// TwinCAT 3 PLC project PLC
// ProgramVersion: 3.1.4023.0
// libraries:
//   Tc2_Standard, * (Beckhoff Automation GmbH)
//   Tc2_System, * (Beckhoff Automation GmbH)
//   Tc3_Module, * (Beckhoff Automation GmbH)
// project tree:
//   / PlcTask.TcTTO
//   POUs/ MAIN.TcPOU
//   DUTs/IO/PDOs/ InfoData_6F19DB2B.TcDUT, CC_Inputs_2C1C9EE0.TcDUT, CC_Outputs_69F9BE14.TcDUT, WcState_9091E0EB.TcDUT, InfoData_BEF6B88E.TcDUT, FB_Inputs_4BC4AA01.TcDUT, FB_Outputs_DAFD38E0.TcDUT, InfoData_A7436BC6.TcDUT, CC_Inputs_14_Ch_F1B79554.TcDUT, CC_Outputs_14_Ch_45965511.TcDUT, FB_Inputs_39145651.TcDUT, FB_Inputs_01C60045.TcDUT, FB_Inputs_2D665851.TcDUT, InfoData_E68C61CD.TcDUT, WcState_0B2B16F9.TcDUT, InfoData_2A97D6CF.TcDUT, Inputs_25A0042B.TcDUT, Outputs_2397A10E.TcDUT
//   DUTs/IO/Boxes/ EK1100_1FC0878B.TcDUT, EK1122_1FC0878B.TcDUT, AT2020_2EA6C9BF.TcDUT, AT2050_33A3DF1B.TcDUT, AT2000_1809CD2F.TcDUT, AT2000_2EA6C9BF.TcDUT, AT2001_2EA6C9BF.TcDUT, AT2002_2EA6C9BF.TcDUT, AT2021_2EA6C9BF.TcDUT, AT2025_2EA6C9BF.TcDUT, AT2026_2EA6C9BF.TcDUT, AT2040_2EA6C9BF.TcDUT, AT2000_33A3DF1B.TcDUT, AT2026_33A3DF1B.TcDUT, AT2041_2EA6C9BF.TcDUT, AT2042_33A3DF1B.TcDUT, AT2041_33A3DF1B.TcDUT, AT2040_33A3DF1B.TcDUT, AT2042_2EA6C9BF.TcDUT, AT2025_33A3DF1B.TcDUT, AT2050_2EA6C9BF.TcDUT, AT2021_33A3DF1B.TcDUT, AT2020_33A3DF1B.TcDUT, AT2001_33A3DF1B.TcDUT, AT2002_33A3DF1B.TcDUT, ATH2000_2EA6C9BF.TcDUT, ATH2050_6EC099B7.TcDUT, ATH2040_41437DDC.TcDUT, ATH2040_2EA6C9BF.TcDUT, ATH2050_2EA6C9BF.TcDUT, ATH2000_D874080E.TcDUT
//   DUTs/IO/Devices/ SyncUnitTask_2D604ED5.TcDUT, SyncUnitTasks_6FEB8257.TcDUT, SyncUnits_99E584AF.TcDUT
//   DUTs/IO/Topology/ A_0060_AT2020_0250_0019_AT2020_0250_29EE8276.TcDUT, A_0036_AT2040_0250_0021_0B822AE4.TcDUT, A_0037_AT2040_0250_0022_033DCEC4.TcDUT, A_0038_AT2040_0250_0023_C339CA0C.TcDUT, A_0039_AT2040_0250_0024_375958EA.TcDUT, A_0040_AT2041_0250_0018_536500F2.TcDUT, A_0041_AT2041_0250_0019_F34F4056.TcDUT, A_0042_AT2041_0250_0020_5E65A51E.TcDUT, A_0043_AT2041_0250_0021_AA0537F8.TcDUT, A_0044_AT2041_0250_0022_5A9A39BA.TcDUT, A_0045_AT2041_0250_0023_51C662AC.TcDUT, A_0046_AT2042_0250_0024_1B20CF31.TcDUT, A_0047_AT2050_0500_0016_139F2B11.TcDUT, A_0048_AT2050_0500_0017_3F977F47.TcDUT, A_0049_AT2050_0500_0018_CBE655A8.TcDUT, A_0050_AT2050_0500_0019_15A3AE6F.TcDUT, A_0051_AT2050_0500_0020_9B531B4E.TcDUT, A_0052_AT2050_0500_0021_4516E089.TcDUT, A_0053_AT2050_0500_0022_433BDDFE.TcDUT, A_0054_AT2050_0500_0023_B2F2DF55.TcDUT, A_0055_AT2050_0500_0024_8D42A08D.TcDUT, A_0056_AT2050_0501_0017_A14AF4DB.TcDUT, A_0057_AT2050_0501_0020_A9F510FB.TcDUT, A_0058_AT2050_0501_0021_DD8E1090.TcDUT, A_0061_AT2020_0250_0023_AT2020_0250_2D9AB3DC.TcDUT, A_0062_AT2025_0250_0020_AT2025_0250_8DB0F378.TcDUT, A_0063_AT2025_0250_0022_AT2025_0250_E88F66A2.TcDUT, A_0064_AT2025_0250_0023_AT2025_0250_894F6FDC.TcDUT, A_0065_AT2026_0250_0019_AT2026_0250_A5473B8A.TcDUT, A_0066_AT2026_0250_0020_AT2026_0250_ADF8DFAA.TcDUT, A_0067_AT2026_0250_0022_AT2026_0250_BF728FE6.TcDUT, A_0068_AT2026_0250_0024_AT2026_0250_71C01165.TcDUT, A_0069_AT2050_0501_0019_AT2050_0501_10255FA6.TcDUT, A_0070_AT2050_0501_0022_AT2050_0501_E445CD40.TcDUT, A_0071_AT2050_0501_0023_AT2050_0501_A5CC9684.TcDUT, A_0072_AT2050_0501_0024_AT2050_0501_05E6D620.TcDUT, Beckhoff_AT2xxxEK1122_43DD63D7.TcDUT, Beckhoff_AT1xxx_27B72169.TcDUT, A_0001_ATH2000_0250_0022_300D1FD0.TcDUT, A_0002_ATH2000_0250_0023_E62B11EA.TcDUT, Beckhoff_ATH2xxxEK1122_61A38CAE.TcDUT, Beckhoff_ATH2xxx_11442560.TcDUT, EtherCAT_Master_ATxxxx_981D2C79.TcDUT
//   DUTs/IO/Base/ EtcSlaveBase_82538BE2.TcDUT, EtcSlaveBase_82538BE2.TcDUT, EtcSlaveBase_82538BE2.TcDUT, EtcSlaveTerminalBase_947E5A46.TcDUT, EtcSlaveBoxBase_77A0E4A7.TcDUT, EtcSlaveEndTerminalBase_866C7F0C.TcDUT, InputBase_8311D824.TcDUT, OutputBase_10CEE7DE.TcDUT, EtcMasterBase_62654B43.TcDUT
//   GVLs/ GVL_iXlinker.TcGVL
// real-time tasks:
//   TASK PlcTask: cycle T#10ms, priority 20, ADS port 350
// I/O:
//   DEVICE EtherCAT_Master_ATxxxx, AmsNetId 172.20.30.238.4.1
//     Beckhoff AT1xxx [EK1100 EtherCAT Coupler (2A E-Bus)]
//       Beckhoff AT2xxxEK1122 [EK1122 2 port EtherCAT junction]
//         A_0060(AT2020-0250-0019) (AT2020-0250) [AT2020-0250 Motor module, +22.5°, 250mm, 50V]
//           A_0085(AT2050-5500-0018) (AT2050-5500) [AT2050-5500 Sensor line 90° clothoid, EtherCAT In]
//         Beckhoff AT2xxxsub EK1100 [EK1100 EtherCAT Coupler (2A E-Bus)]
//         A_0001(AT2000-0233-0022) [AT2000-0233 Motor module 233 mm, 48V]
//         A_0002(AT2000-0233-0023) [AT2000-0233 Motor module 233 mm, 48V]
//         A_0003(AT2000-0233-0024) [AT2000-0233 Motor module 233 mm, 48V]
//         A_0004(AT2000-0250-0016) [AT2000-0250 Motor module 250 mm, 50V]
//         A_0005(AT2000-0250-0017) [AT2000-0250 Motor module 250 mm, 50V]
//         A_0006(AT2000-0250-0018) [AT2000-0250 Motor module 250 mm, 50V]
//         A_0007(AT2000-0250-0019) [AT2000-0250 Motor module 250 mm, 50V]
//         A_0008(AT2000-0250-0020) [AT2000-0250 Motor module 250 mm, 48V]
//         A_0009(AT2000-0250-0021) [AT2000-0250 Motor module 250 mm, 48V]
//         A_0010(AT2000-0250-0022) [AT2000-0250 Motor module 250 mm, 48V]
//         A_0011(AT2000-0250-0023) [AT2000-0250 Motor module 250 mm, 48V]
//         A_0012(AT2001-0250-0016) [AT2001-0250 Motor module with feed 250 mm, 50V]
//         A_0013(AT2001-0250-0017) [AT2001-0250 Motor module with feed 250 mm, 50V]
//         A_0014(AT2001-0250-0018) [AT2001-0250 Motor module with feed 250 mm, 50V]
//         A_0015(AT2001-0250-0019) [AT2001-0250 Motor module with feed 250 mm, 50V]
//         A_0016(AT2001-0250-0020) [AT2001-0250 Motor module with feed 250 mm, 48V]
//         A_0017(AT2001-0250-0022) [AT2001-0250 Motor module with feed 250 mm, 48V]
//         A_0018(AT2001-0250-0023) [AT2001-0250 Motor module with feed 250 mm, 48V]
//         A_0019(AT2001-0250-0024) [AT2001-0250 Motor module with feed 250 mm, 48V]
//         A_0020(AT2002-0249-0021) [AT2002-0249 Motor module (Track management) with feed 249 mm, 48V]
//         A_0021(AT2002-0249-0022) [AT2002-0249 Motor module (Track management) with feed 249 mm, 48V]
//         A_0022(AT2002-0249-0023) [AT2002-0249 Motor module (Track management) with feed 249 mm, 48V]
//         A_0023(AT2002-0250-0022) [AT2002-0250 Motor module with feed (B23-Connector), 250 mm, 48V]
//         A_0024(AT2002-0250-0023) [AT2002-0250 Motor module with feed (B23-Connector) 250 mm, 48V]
//         A_0025(AT2002-0250-0024) [AT2002-0250 Motor module with feed (B23-Connector) 250 mm, 48V]
//         A_0026(AT2020-0250-0018) [AT2020-0250 Motor module, +22.5°, 250mm, 50V]
//         A_0027(AT2020-0250-0021) [AT2020-0250 Motor module, +22.5°, 250mm, 48V]
//         A_0028(AT2021-0250-0018) [AT2021-0250 Motor module with feed , +22.5°, 250mm, 50V]
//         A_0029(AT2021-0250-0020) [AT2021-0250 Motor module with feed , +22.5°, 250mm, 48V]
//         A_0030(AT2025-0250-0018) [AT2025-0250 Motor module, -22.5°, 250mm, 50V]
//         A_0031(AT2026-0250-0021) [AT2026-0250 Motor module with feed, -22.5°, 250mm, 48V]
//         A_0032(AT2026-0250-0023) [AT2026-0250 Motor module with feed, -22.5°, 250mm, 48V]
//         A_0033(AT2040-0250-0018) [AT2040-0250 Motor module, +45°, 250mm, 50V]
//         A_0034(AT2040-0250-0019) [AT2040-0250 Motor module, +45°, 250mm, 50V]
//         A_0035(AT2040-0250-0020) [AT2040-0250 Motor module, +45°, 250mm, 48V]
//         A_0036(AT2040-0250-0021) [AT2040-0250 Motor module, +45°, 250mm, 48V]
//           A_0108(AT2000-5233-0019) (AT2000-5233) [AT2000-5233 Sensor line 233 mm]
//         A_0037(AT2040-0250-0022) [AT2040-0250 Motor module, +45°, 250mm, 48V]
//           A_0107(AT2000-5233-0018) (AT2000-5233) [AT2000-5233 Sensor line 233 mm]
//         A_0038(AT2040-0250-0023) [AT2040-0250 Motor module, +45°, 250mm, 48V]
//           A_0106(AT2026-5250-0019) (AT2026-5250) [AT2026-5250 Sensor line with feed, -22.5°]
//         A_0039(AT2040-0250-0024) [AT2040-0250 Motor module, +45°, 250mm, 48V]
//           A_0105(AT2026-5250-0018) (AT2026-5250) [AT2026-5250 Sensor line with feed, -22.5°]
//         A_0040(AT2041-0250-0018) [AT2041-0250 Motor module with feed, +45°, 250mm, 50V]
//           A_0104(AT2042-5250-0019) (AT2042-5250) [AT2042-5250 Sensor line with feed (B23-Connector), +45°]
//         A_0041(AT2041-0250-0019) [AT2041-0250 Motor module with feed, +45°, 250mm, 50V]
//           A_0103(AT2042-5250-0018) (AT2042-5250) [AT2042-5250 Sensor line with feed (B23-Connector), +45°]
//         A_0042(AT2041-0250-0020) [AT2041-0250 Motor module with feed, +45°, 250mm, 48V]
//           A_0102(AT2041-5250-0019) (AT2041-5250) [AT2041-5250 Sensor line with feed, +45°]
//         A_0043(AT2041-0250-0021) [AT2041-0250 Motor module with feed, +45°, 250mm, 48V]
//           A_0101(AT2041-5250-0018) (AT2041-5250) [AT2041-5250 Sensor line with feed, +45°]
//         A_0044(AT2041-0250-0022) [AT2041-0250 Motor module with feed, +45°, 250mm, 48V]
//           A_0100(AT2040-5250-0019) (AT2040-5250) [AT2040-5250 Sensor line +45°]
//         A_0045(AT2041-0250-0023) [AT2041-0250 Motor module with feed, +45°, 250mm, 48V]
//           A_0099(AT2040-5250-0018) (AT2040-5250) [AT2040-5250 Sensor line +45°]
//         A_0046(AT2042-0250-0024) [AT2042-0250 Motor module with feed (B23-Connector), +45°, 250 mm, 48V]
//           A_0098(AT2025-5250-0019) (AT2025-5250) [AT2025-5250 Sensor line -22.5°]
//         A_0047(AT2050-0500-0016) [AT2050-0500 Motor module, 90° clothoid, EtherCAT In, 50V]
//           A_0097(AT2025-5250-0018) (AT2025-5250) [AT2025-5250 Sensor line -22.5°]
//         A_0048(AT2050-0500-0017) [AT2050-0500 Motor module, 90° clothoid, EtherCAT In, 50V]
//           A_0096(AT2025-5250-0017) (AT2025-5250) [AT2025-5250 Sensor line -22.5°]
//         A_0049(AT2050-0500-0018) [AT2050-0500 Motor module, 90° clothoid, EtherCAT In, 50V]
//           A_0095(AT2021-5250-0019) (AT2021-5250) [AT2021-5250 Sensor line with feed, +22.5°]
//         A_0050(AT2050-0500-0019) [AT2050-0500 Motor module, 90° clothoid, EtherCAT In, 50V]
//           A_0094(AT2021-5250-0018) (AT2021-5250) [AT2021-5250 Sensor line with feed, +22.5°]
//         A_0051(AT2050-0500-0020) [AT2050-0500 Motor module, 90° clothoid, EtherCAT In, 48V]
//           A_0093(AT2020-5250-0019) (AT2020-5250) [AT2020-5250 Sensor line +22.5°]
//         A_0052(AT2050-0500-0021) [AT2050-0500 Motor module, 90° clothoid, EtherCAT In, 48V]
//           A_0092(AT2020-5250-0018) (AT2020-5250) [AT2020-5250 Sensor line +22.5°]
//         A_0053(AT2050-0500-0022) [AT2050-0500 Motor module, 90° clothoid, EtherCAT In, 48V]
//           A_0091(AT2020-5250-0017) (AT2020-5250) [AT2020-5250 Sensor line +22.5°]
//         A_0054(AT2050-0500-0023) [AT2050-0500 Motor module, 90° clothoid, EtherCAT In, 48V]
//           A_0090(AT2050-5501-0019) (AT2050-5501) [AT2050-5501 Sensor line 90° clothoid, EtherCAT Out]
//         A_0055(AT2050-0500-0024) [AT2050-0500 Motor module, 90° clothoid, EtherCAT In, 48V]
//           A_0089(AT2050-5501-0018) (AT2050-5501) [AT2050-5501 Sensor line 90° clothoid, EtherCAT Out]
//         A_0056(AT2050-0501-0017) [AT2050-0501 Motor module, 90° clothoid, EtherCAT Out, 50V]
//           A_0088(AT2050-5501-0017) (AT2050-5501) [AT2050-5501 Sensor line 90° clothoid, EtherCAT Out]
//         A_0057(AT2050-0501-0020) [AT2050-0501 Motor module, 90° clothoid, EtherCAT Out, 48V]
//           A_0087(AT2050-5501-0016) (AT2050-5501) [AT2050-5501 Sensor line 90° clothoid, EtherCAT Out]
//         A_0058(AT2050-0501-0021) [AT2050-0501 Motor module, 90° clothoid, EtherCAT Out, 48V]
//           A_0086(AT2050-5500-0019) (AT2050-5500) [AT2050-5500 Sensor line 90° clothoid, EtherCAT In]
//         A_0061(AT2020-0250-0023) (AT2020-0250) [AT2020-0250 Motor module, +22.5°, 250mm, 48V]
//           A_0073(AT2000-5250-0016) (AT2000-5250) [AT2000-5250 Sensor line]
//         A_0062(AT2025-0250-0020) (AT2025-0250) [AT2025-0250 Motor module, -22.5°, 250mm, 48V]
//           A_0074(AT2000-5250-0017) (AT2000-5250) [AT2000-5250 Sensor line]
//         A_0063(AT2025-0250-0022) (AT2025-0250) [AT2025-0250 Motor module, -22.5°, 250mm, 48V]
//           A_0075(AT2000-5250-0019) (AT2000-5250) [AT2000-5250 Sensor line]
//         A_0064(AT2025-0250-0023) (AT2025-0250) [AT2025-0250 Motor module, -22.5°, 250mm, 48V]
//           A_0076(AT2001-5250-0017) (AT2001-5250) [AT2001-5250 Sensor line with feed]
//         A_0065(AT2026-0250-0019) (AT2026-0250) [AT2026-0250 Motor module with feed, -22.5°, 250mm, 50V]
//           A_0077(AT2001-5250-0018) (AT2001-5250) [AT2001-5250 Sensor line with feed]
//         A_0066(AT2026-0250-0020) (AT2026-0250) [AT2026-0250 Motor module with feed, -22.5°, 250mm, 48V]
//           A_0078(AT2001-5250-0019) (AT2001-5250) [AT2001-5250 Sensor line with feed]
//         A_0067(AT2026-0250-0022) (AT2026-0250) [AT2026-0250 Motor module with feed, -22.5°, 250mm, 48V]
//           A_0079(AT2002-5249-0018) (AT2002-5249) [AT2002-5249 Sensor line (Track management) with feed]
//         A_0068(AT2026-0250-0024) (AT2026-0250) [AT2026-0250 Motor module with feed, -22.5°, 250mm, 48V]
//           A_0080(AT2002-5249-0019) (AT2002-5249) [AT2002-5249 Sensor line (Track management) with feed]
//         A_0069(AT2050-0501-0019) (AT2050-0501) [AT2050-0501 Motor module, 90° clothoid, EtherCAT Out, 50V]
//           A_0081(AT2002-5250-0018) (AT2002-5250) [AT2002-5250 Sensor line with feed (B23-Connector)]
//         A_0070(AT2050-0501-0022) (AT2050-0501) [AT2050-0501 Motor module, 90° clothoid, EtherCAT Out, 48V]
//           A_0082(AT2002-5250-0019) (AT2002-5250) [AT2002-5250 Sensor line with feed (B23-Connector)]
//         A_0071(AT2050-0501-0023) (AT2050-0501) [AT2050-0501 Motor module, 90° clothoid, EtherCAT Out, 48V]
//           A_0083(AT2050-5500-0016) (AT2050-5500) [AT2050-5500 Sensor line 90° clothoid, EtherCAT In]
//         A_0072(AT2050-0501-0024) (AT2050-0501) [AT2050-0501 Motor module, 90° clothoid, EtherCAT Out, 48V]
//           A_0084(AT2050-5500-0017) (AT2050-5500) [AT2050-5500 Sensor line 90° clothoid, EtherCAT In]
//       A_0059(AT2000-5250-0018) [AT2000-5250 Sensor line]
//     Beckhoff ATH2xxx [EK1100 EtherCAT Coupler (2A E-Bus)]
//       Beckhoff ATH2xxxEK1122 [EK1122 2 port EtherCAT junction]
//         Beckhoff ATH2xxxsub EK1100 [EK1100 EtherCAT Coupler (2A E-Bus)]
//         A_0001(ATH2000-0250-0022) [ATH2000-0250 Hygienic Motor module 250 mm, 48V]
//           A_0014(ATH2050-5501-0022) [ATH2050-5501 Hygienic Sensor 90° clothoid, EtherCAT Out]
//         A_0002(ATH2000-0250-0023) [ATH2000-0250 Hygienic Motor module 250 mm, 48V]
//           A_0015(ATH2040-5250-0022) [ATH2040-5250 Hygienic Sensor +45°]
//         A_0003(ATH2000-0250-0024) [ATH2000-0250 Hygienic Motor module 250 mm, 48V]
//         A_0004(ATH2040-0250-0022) [ATH2040-0250 Hygienic Motor module +45°, 250mm, 48V]
//         A_0005(ATH2040-0250-0023) [ATH2040-0250 Hygienic Motor module +45°, 250mm, 48V]
//         A_0006(ATH2040-0250-0024) [ATH2040-0250 Hygienic Motor module +45°, 250mm, 48V]
//         A_0007(ATH2050-0500-0022) [ATH2050-0500 Hygienic Motor module 90° clothoid, EtherCAT In]
//         A_0008(ATH2050-0500-0023) [ATH2050-0500 Hygienic Motor module 90° clothoid, EtherCAT In]
//         A_0009(ATH2050-0500-0024) [ATH2050-0500 Hygienic Motor module 90° clothoid, EtherCAT In]
//         A_0010(ATH2050-0501-0022) [ATH2050-0501 Hygienic Motor module 90° clothoid, EtherCAT Out]
//         A_0011(ATH2050-0501-0023) [ATH2050-0501 Hygienic Motor module 90° clothoid, EtherCAT Out]
//         A_0012(ATH2050-0501-0024) [ATH2050-0501 Hygienic Motor module 90° clothoid, EtherCAT Out]
//       A_0013(ATH2000-5250-0022) [ATH2000-5250 Hygienic Sensor line]
// variable links:
//   PLC/PLC Instance <-> EtherCAT Master ATxxxx/Beckhoff AT1xxx
//     PlcTask Inputs/GVL_iXlinker.EtherCAT_Master_ATxxxx.Beckhoff_AT1xxx.InfoData.State <-> InfoData/State
//   PLC/PLC Instance <-> EtherCAT Master ATxxxx/Beckhoff AT1xxx/Beckhoff AT2xxxEK1122
//     PlcTask Inputs/GVL_iXlinker.EtherCAT_Master_ATxxxx.Beckhoff_AT1xxx.Beckhoff_AT2xxxEK1122.InfoData.State <-> InfoData/State
//   PLC/PLC Instance <-> EtherCAT Master ATxxxx/Beckhoff AT1xxx/Beckhoff AT2xxxEK1122/A_0060(AT2020-0250-0019) (AT2020-0250)
//     PlcTask Inputs/GVL_iXlinker.EtherCAT_Master_ATxxxx.Beckhoff_AT1xxx.Beckhoff_AT2xxxEK1122.A_0060_AT2020_0250_0019_AT2020_0250.CC_Inputs.Status <-> CC Inputs/Status
//     PlcTask Inputs/GVL_iXlinker.EtherCAT_Master_ATxxxx.Beckhoff_AT1xxx.Beckhoff_AT2xxxEK1122.A_0060_AT2020_0250_0019_AT2020_0250.CC_Inputs.Current_actual_value_Ch[0] <-> CC Inputs/Current actual value Ch.1
//     PlcTask Inputs/GVL_iXlinker.EtherCAT_Master_ATxxxx.Beckhoff_AT1xxx.Beckhoff_AT2xxxEK1122.A_0060_AT2020_0250_0019_AT2020_0250.CC_Inputs.Current_actual_value_Ch[1] <-> CC Inputs/Current actual value Ch.2
//     PlcTask Inputs/GVL_iXlinker.EtherCAT_Master_ATxxxx.Beckhoff_AT1xxx.Beckhoff_AT2xxxEK1122.A_0060_AT2020_0250_0019_AT2020_0250.CC_Inputs.Current_actual_value_Ch[2] <-> CC Inputs/Current actual value Ch.3
//     PlcTask Inputs/GVL_iXlinker.EtherCAT_Master_ATxxxx.Beckhoff_AT1xxx.Beckhoff_AT2xxxEK1122.A_0060_AT2020_0250_0019_AT2020_0250.CC_Inputs.Current_actual_value_Ch[3] <-> CC Inputs/Current actual value Ch.4
//     PlcTask Inputs/GVL_iXlinker.EtherCAT_Master_ATxxxx.Beckhoff_AT1xxx.Beckhoff_AT2xxxEK1122.A_0060_AT2020_0250_0019_AT2020_0250.CC_Inputs.Current_actual_value_Ch[4] <-> CC Inputs/Current actual value Ch.5
//     PlcTask Inputs/GVL_iXlinker.EtherCAT_Master_ATxxxx.Beckhoff_AT1xxx.Beckhoff_AT2xxxEK1122.A_0060_AT2020_0250_0019_AT2020_0250.CC_Inputs.Current_actual_value_Ch[5] <-> CC Inputs/Current actual value Ch.6
//     PlcTask Inputs/GVL_iXlinker.EtherCAT_Master_ATxxxx.Beckhoff_AT1xxx.Beckhoff_AT2xxxEK1122.A_0060_AT2020_0250_0019_AT2020_0250.CC_Inputs.Current_actual_value_Ch[6] <-> CC Inputs/Current actual value Ch.7
//     PlcTask Inputs/GVL_iXlinker.EtherCAT_Master_ATxxxx.Beckhoff_AT1xxx.Beckhoff_AT2xxxEK1122.A_0060_AT2020_0250_0019_AT2020_0250.CC_Inputs.Current_actual_value_Ch[7] <-> CC Inputs/Current actual value Ch.8
//     PlcTask Inputs/GVL_iXlinker.EtherCAT_Master_ATxxxx.Beckhoff_AT1xxx.Beckhoff_AT2xxxEK1122.A_0060_AT2020_0250_0019_AT2020_0250.CC_Inputs.Current_actual_value_Ch[8] <-> CC Inputs/Current actual value Ch.9
//     PlcTask Inputs/GVL_iXlinker.EtherCAT_Master_ATxxxx.Beckhoff_AT1xxx.Beckhoff_AT2xxxEK1122.A_0060_AT2020_0250_0019_AT2020_0250.CC_Inputs.Current_actual_value_Ch[9] <-> CC Inputs/Current actual value Ch.10
//     PlcTask Inputs/GVL_iXlinker.EtherCAT_Master_ATxxxx.Beckhoff_AT1xxx.Beckhoff_AT2xxxEK1122.A_0060_AT2020_0250_0019_AT2020_0250.CC_Inputs.Current_actual_value_Ch[10] <-> CC Inputs/Current actual value Ch.11
//     PlcTask Inputs/GVL_iXlinker.EtherCAT_Master_ATxxxx.Beckhoff_AT1xxx.Beckhoff_AT2xxxEK1122.A_0060_AT2020_0250_0019_AT2020_0250.CC_Inputs.Current_actual_value_Ch[11] <-> CC Inputs/Current actual value Ch.12
//     PlcTask Inputs/GVL_iXlinker.EtherCAT_Master_ATxxxx.Beckhoff_AT1xxx.Beckhoff_AT2xxxEK1122.A_0060_AT2020_0250_0019_AT2020_0250.CC_Inputs.Current_actual_value_Ch[12] <-> CC Inputs/Current actual value Ch.13
//     PlcTask Inputs/GVL_iXlinker.EtherCAT_Master_ATxxxx.Beckhoff_AT1xxx.Beckhoff_AT2xxxEK1122.A_0060_AT2020_0250_0019_AT2020_0250.CC_Inputs.Current_actual_value_Ch[13] <-> CC Inputs/Current actual value Ch.14
//     PlcTask Inputs/GVL_iXlinker.EtherCAT_Master_ATxxxx.Beckhoff_AT1xxx.Beckhoff_AT2xxxEK1122.A_0060_AT2020_0250_0019_AT2020_0250.CC_Inputs.Current_actual_value_Ch[14] <-> CC Inputs/Current actual value Ch.15
//     PlcTask Outputs/GVL_iXlinker.EtherCAT_Master_ATxxxx.Beckhoff_AT1xxx.Beckhoff_AT2xxxEK1122.A_0060_AT2020_0250_0019_AT2020_0250.CC_Outputs.Control <-> CC Outputs/Control
//     PlcTask Outputs/GVL_iXlinker.EtherCAT_Master_ATxxxx.Beckhoff_AT1xxx.Beckhoff_AT2xxxEK1122.A_0060_AT2020_0250_0019_AT2020_0250.CC_Outputs.Current_setpoint_value_Ch[0] <-> CC Outputs/Current setpoint value Ch.1
//     PlcTask Outputs/GVL_iXlinker.EtherCAT_Master_ATxxxx.Beckhoff_AT1xxx.Beckhoff_AT2xxxEK1122.A_0060_AT2020_0250_0019_AT2020_0250.CC_Outputs.Current_setpoint_value_Ch[1] <-> CC Outputs/Current setpoint value Ch.2
//     PlcTask Outputs/GVL_iXlinker.EtherCAT_Master_ATxxxx.Beckhoff_AT1xxx.Beckhoff_AT2xxxEK1122.A_0060_AT2020_0250_0019_AT2020_0250.CC_Outputs.Current_setpoint_value_Ch[2] <-> CC Outputs/Current setpoint value Ch.3
//     PlcTask Outputs/GVL_iXlinker.EtherCAT_Master_ATxxxx.Beckhoff_AT1xxx.Beckhoff_AT2xxxEK1122.A_0060_AT2020_0250_0019_AT2020_0250.CC_Outputs.Current_setpoint_value_Ch[3] <-> CC Outputs/Current setpoint value Ch.4
//     PlcTask Outputs/GVL_iXlinker.EtherCAT_Master_ATxxxx.Beckhoff_AT1xxx.Beckhoff_AT2xxxEK1122.A_0060_AT2020_0250_0019_AT2020_0250.CC_Outputs.Current_setpoint_value_Ch[4] <-> CC Outputs/Current setpoint value Ch.5
//     PlcTask Outputs/GVL_iXlinker.EtherCAT_Master_ATxxxx.Beckhoff_AT1xxx.Beckhoff_AT2xxxEK1122.A_0060_AT2020_0250_0019_AT2020_0250.CC_Outputs.Current_setpoint_value_Ch[5] <-> CC Outputs/Current setpoint value Ch.6
//     PlcTask Outputs/GVL_iXlinker.EtherCAT_Master_ATxxxx.Beckhoff_AT1xxx.Beckhoff_AT2xxxEK1122.A_0060_AT2020_0250_0019_AT2020_0250.CC_Outputs.Current_setpoint_value_Ch[6] <-> CC Outputs/Current setpoint value Ch.7
//     PlcTask Outputs/GVL_iXlinker.EtherCAT_Master_ATxxxx.Beckhoff_AT1xxx.Beckhoff_AT2xxxEK1122.A_0060_AT2020_0250_0019_AT2020_0250.CC_Outputs.Current_setpoint_value_Ch[7] <-> CC Outputs/Current setpoint value Ch.8
//     PlcTask Outputs/GVL_iXlinker.EtherCAT_Master_ATxxxx.Beckhoff_AT1xxx.Beckhoff_AT2xxxEK1122.A_0060_AT2020_0250_0019_AT2020_0250.CC_Outputs.Current_setpoint_value_Ch[8] <-> CC Outputs/Current setpoint value Ch.9
//     PlcTask Outputs/GVL_iXlinker.EtherCAT_Master_ATxxxx.Beckhoff_AT1xxx.Beckhoff_AT2xxxEK1122.A_0060_AT2020_0250_0019_AT2020_0250.CC_Outputs.Current_setpoint_value_Ch[9] <-> CC Outputs/Current setpoint value Ch.10
//     PlcTask Outputs/GVL_iXlinker.EtherCAT_Master_ATxxxx.Beckhoff_AT1xxx.Beckhoff_AT2xxxEK1122.A_0060_AT2020_0250_0019_AT2020_0250.CC_Outputs.Current_setpoint_value_Ch[10] <-> CC Outputs/Current setpoint value Ch.11
//     PlcTask Outputs/GVL_iXlinker.EtherCAT_Master_ATxxxx.Beckhoff_AT1xxx.Beckhoff_AT2xxxEK1122.A_0060_AT2020_0250_0019_AT2020_0250.CC_Outputs.Current_setpoint_value_Ch[11] <-> CC Outputs/Current setpoint value Ch.12
//     PlcTask Outputs/GVL_iXlinker.EtherCAT_Master_ATxxxx.Beckhoff_AT1xxx.Beckhoff_AT2xxxEK1122.A_0060_AT2020_0250_0019_AT2020_0250.CC_Outputs.Current_setpoint_value_Ch[12] <-> CC Outputs/Current setpoint value Ch.13
//     PlcTask Outputs/GVL_iXlinker.EtherCAT_Master_ATxxxx.Beckhoff_AT1xxx.Beckhoff_AT2xxxEK1122.A_0060_AT2020_0250_0019_AT2020_0250.CC_Outputs.Current_setpoint_value_Ch[13] <-> CC Outputs/Current setpoint value Ch.14
//     PlcTask Outputs/GVL_iXlinker.EtherCAT_Master_ATxxxx.Beckhoff_AT1xxx.Beckhoff_AT2xxxEK1122.A_0060_AT2020_0250_0019_AT2020_0250.CC_Outputs.Current_setpoint_value_Ch[14] <-> CC Outputs/Current setpoint value Ch.15
//     PlcTask Inputs/GVL_iXlinker.EtherCAT_Master_ATxxxx.Beckhoff_AT1xxx.Beckhoff_AT2xxxEK1122.A_0060_AT2020_0250_0019_AT2020_0250.WcState.WcState <-> WcState/WcState
//     PlcTask Inputs/GVL_iXlinker.EtherCAT_Master_ATxxxx.Beckhoff_AT1xxx.Beckhoff_AT2xxxEK1122.A_0060_AT2020_0250_0019_AT2020_0250.WcState.InputToggle <-> WcState/InputToggle
//     PlcTask Inputs/GVL_iXlinker.EtherCAT_Master_ATxxxx.Beckhoff_AT1xxx.Beckhoff_AT2xxxEK1122.A_0060_AT2020_0250_0019_AT2020_0250.InfoData.AdsAddr <-> InfoData/AdsAddr
//     PlcTask Inputs/GVL_iXlinker.EtherCAT_Master_ATxxxx.Beckhoff_AT1xxx.Beckhoff_AT2xxxEK1122.A_0060_AT2020_0250_0019_AT2020_0250.InfoData.DcOutputShift <-> InfoData/DcOutputShift
//     PlcTask Inputs/GVL_iXlinker.EtherCAT_Master_ATxxxx.Beckhoff_AT1xxx.Beckhoff_AT2xxxEK1122.A_0060_AT2020_0250_0019_AT2020_0250.InfoData.DcInputShift <-> InfoData/DcInputShift
//     PlcTask Inputs/GVL_iXlinker.EtherCAT_Master_ATxxxx.Beckhoff_AT1xxx.Beckhoff_AT2xxxEK1122.A_0060_AT2020_0250_0019_AT2020_0250.InfoData.State <-> InfoData/State
//   PLC/PLC Instance <-> EtherCAT Master ATxxxx/Beckhoff AT1xxx/Beckhoff AT2xxxEK1122/A_0060(AT2020-0250-0019) (AT2020-0250)/A_0085(AT2050-5500-0018) (AT2050-5500)
//     PlcTask Inputs/GVL_iXlinker.EtherCAT_Master_ATxxxx.Beckhoff_AT1xxx.Beckhoff_AT2xxxEK1122.A_0060_AT2020_0250_0019_AT2020_0250.A_0085_AT2050_5500_0018_AT2050_5500.FB_Inputs.Status <-> FB Inputs/Status
//     PlcTask Inputs/GVL_iXlinker.EtherCAT_Master_ATxxxx.Beckhoff_AT1xxx.Beckhoff_AT2xxxEK1122.A_0060_AT2020_0250_0019_AT2020_0250.A_0085_AT2050_5500_0018_AT2050_5500.FB_Inputs.Value_Channel[0] <-> FB Inputs/Value Channel 01
//     PlcTask Inputs/GVL_iXlinker.EtherCAT_Master_ATxxxx.Beckhoff_AT1xxx.Beckhoff_AT2xxxEK1122.A_0060_AT2020_0250_0019_AT2020_0250.A_0085_AT2050_5500_0018_AT2050_5500.FB_Inputs.Value_Channel[1] <-> FB Inputs/Value Channel 02
//     PlcTask Inputs/GVL_iXlinker.EtherCAT_Master_ATxxxx.Beckhoff_AT1xxx.Beckhoff_AT2xxxEK1122.A_0060_AT2020_0250_0019_AT2020_0250.A_0085_AT2050_5500_0018_AT2050_5500.FB_Inputs.Value_Channel[2] <-> FB Inputs/Value Channel 03
//     PlcTask Inputs/GVL_iXlinker.EtherCAT_Master_ATxxxx.Beckhoff_AT1xxx.Beckhoff_AT2xxxEK1122.A_0060_AT2020_0250_0019_AT2020_0250.A_0085_AT2050_5500_0018_AT2050_5500.FB_Inputs.Value_Channel[3] <-> FB Inputs/Value Channel 04
//     PlcTask Inputs/GVL_iXlinker.EtherCAT_Master_ATxxxx.Beckhoff_AT1xxx.Beckhoff_AT2xxxEK1122.A_0060_AT2020_0250_0019_AT2020_0250.A_0085_AT2050_5500_0018_AT2050_5500.FB_Inputs.Value_Channel[4] <-> FB Inputs/Value Channel 05
//     PlcTask Inputs/GVL_iXlinker.EtherCAT_Master_ATxxxx.Beckhoff_AT1xxx.Beckhoff_AT2xxxEK1122.A_0060_AT2020_0250_0019_AT2020_0250.A_0085_AT2050_5500_0018_AT2050_5500.FB_Inputs.Value_Channel[5] <-> FB Inputs/Value Channel 06
//     PlcTask Inputs/GVL_iXlinker.EtherCAT_Master_ATxxxx.Beckhoff_AT1xxx.Beckhoff_AT2xxxEK1122.A_0060_AT2020_0250_0019_AT2020_0250.A_0085_AT2050_5500_0018_AT2050_5500.FB_Inputs.Value_Channel[6] <-> FB Inputs/Value Channel 07
//     PlcTask Inputs/GVL_iXlinker.EtherCAT_Master_ATxxxx.Beckhoff_AT1xxx.Beckhoff_AT2xxxEK1122.A_0060_AT2020_0250_0019_AT2020_0250.A_0085_AT2050_5500_0018_AT2050_5500.FB_Inputs.Value_Channel[7] <-> FB Inputs/Value Channel 08
//     PlcTask Inputs/GVL_iXlinker.EtherCAT_Master_ATxxxx.Beckhoff_AT1xxx.Beckhoff_AT2xxxEK1122.A_0060_AT2020_0250_0019_AT2020_0250.A_0085_AT2050_5500_0018_AT2050_5500.FB_Inputs.Value_Channel[8] <-> FB Inputs/Value Channel 09
//     PlcTask Inputs/GVL_iXlinker.EtherCAT_Master_ATxxxx.Beckhoff_AT1xxx.Beckhoff_AT2xxxEK1122.A_0060_AT2020_0250_0019_AT2020_0250.A_0085_AT2050_5500_0018_AT2050_5500.FB_Inputs.Value_Channel[9] <-> FB Inputs/Value Channel 10
//     PlcTask Inputs/GVL_iXlinker.EtherCAT_Master_ATxxxx.Beckhoff_AT1xxx.Beckhoff_AT2xxxEK1122.A_0060_AT2020_0250_0019_AT2020_0250.A_0085_AT2050_5500_0018_AT2050_5500.FB_Inputs.Value_Channel[10] <-> FB Inputs/Value Channel 11
//     PlcTask Inputs/GVL_iXlinker.EtherCAT_Master_ATxxxx.Beckhoff_AT1xxx.Beckhoff_AT2xxxEK1122.A_0060_AT2020_0250_0019_AT2020_0250.A_0085_AT2050_5500_0018_AT2050_5500.FB_Inputs.Value_Channel[11] <-> FB Inputs/Value Channel 12
//     PlcTask Inputs/GVL_iXlinker.EtherCAT_Master_ATxxxx.Beckhoff_AT1xxx.Beckhoff_AT2xxxEK1122.A_0060_AT2020_0250_0019_AT2020_0250.A_0085_AT2050_5500_0018_AT2050_5500.FB_Inputs.Value_Channel[12] <-> FB Inputs/Value Channel 13
//     PlcTask Inputs/GVL_iXlinker.EtherCAT_Master_ATxxxx.Beckhoff_AT1xxx.Beckhoff_AT2xxxEK1122.A_0060_AT2020_0250_0019_AT2020_0250.A_0085_AT2050_5500_0018_AT2050_5500.FB_Inputs.Value_Channel[13] <-> FB Inputs/Value Channel 14
//     PlcTask Inputs/GVL_iXlinker.EtherCAT_Master_ATxxxx.Beckhoff_AT1xxx.Beckhoff_AT2xxxEK1122.A_0060_AT2020_0250_0019_AT2020_0250.A_0085_AT2050_5500_0018_AT2050_5500.FB_Inputs.Value_Channel[14] <-> FB Inputs/Value Channel 15
//     PlcTask Inputs/GVL_iXlinker.EtherCAT_Master_ATxxxx.Beckhoff_AT1xxx.Beckhoff_AT2xxxEK1122.A_0060_AT2020_0250_0019_AT2020_0250.A_0085_AT2050_5500_0018_AT2050_5500.FB_Inputs.Value_Channel[15] <-> FB Inputs/Value Channel 16
//     PlcTask Inputs/GVL_iXlinker.EtherCAT_Master_ATxxxx.Beckhoff_AT1xxx.Beckhoff_AT2xxxEK1122.A_0060_AT2020_0250_0019_AT2020_0250.A_0085_AT2050_5500_0018_AT2050_5500.FB_Inputs.Value_Channel[16] <-> FB Inputs/Value Channel 17
//     PlcTask Inputs/GVL_iXlinker.EtherCAT_Master_ATxxxx.Beckhoff_AT1xxx.Beckhoff_AT2xxxEK1122.A_0060_AT2020_0250_0019_AT2020_0250.A_0085_AT2050_5500_0018_AT2050_5500.FB_Inputs.Value_Channel[17] <-> FB Inputs/Value Channel 18
//     PlcTask Inputs/GVL_iXlinker.EtherCAT_Master_ATxxxx.Beckhoff_AT1xxx.Beckhoff_AT2xxxEK1122.A_0060_AT2020_0250_0019_AT2020_0250.A_0085_AT2050_5500_0018_AT2050_5500.FB_Inputs.Value_Channel[18] <-> FB Inputs/Value Channel 19
//     PlcTask Inputs/GVL_iXlinker.EtherCAT_Master_ATxxxx.Beckhoff_AT1xxx.Beckhoff_AT2xxxEK1122.A_0060_AT2020_0250_0019_AT2020_0250.A_0085_AT2050_5500_0018_AT2050_5500.FB_Inputs.Value_Channel[19] <-> FB Inputs/Value Channel 20
//     PlcTask Inputs/GVL_iXlinker.EtherCAT_Master_ATxxxx.Beckhoff_AT1xxx.Beckhoff_AT2xxxEK1122.A_0060_AT2020_0250_0019_AT2020_0250.A_0085_AT2050_5500_0018_AT2050_5500.FB_Inputs.Value_Channel[20] <-> FB Inputs/Value Channel 21
//     PlcTask Inputs/GVL_iXlinker.EtherCAT_Master_ATxxxx.Beckhoff_AT1xxx.Beckhoff_AT2xxxEK1122.A_0060_AT2020_0250_0019_AT2020_0250.A_0085_AT2050_5500_0018_AT2050_5500.FB_Inputs.Value_Channel[21] <-> FB Inputs/Value Channel 22
//     PlcTask Inputs/GVL_iXlinker.EtherCAT_Master_ATxxxx.Beckhoff_AT1xxx.Beckhoff_AT2xxxEK1122.A_0060_AT2020_0250_0019_AT2020_0250.A_0085_AT2050_5500_0018_AT2050_5500.FB_Inputs.Value_Channel[22] <-> FB Inputs/Value Channel 23
//     PlcTask Inputs/GVL_iXlinker.EtherCAT_Master_ATxxxx.Beckhoff_AT1xxx.Beckhoff_AT2xxxEK1122.A_0060_AT2020_0250_0019_AT2020_0250.A_0085_AT2050_5500_0018_AT2050_5500.FB_Inputs.Value_Channel[23] <-> FB Inputs/Value Channel 24
//     PlcTask Inputs/GVL_iXlinker.EtherCAT_Master_ATxxxx.Beckhoff_AT1xxx.Beckhoff_AT2xxxEK1122.A_0060_AT2020_0250_0019_AT2020_0250.A_0085_AT2050_5500_0018_AT2050_5500.FB_Inputs.Value_Channel[24] <-> FB Inputs/Value Channel 25
//     PlcTask Inputs/GVL_iXlinker.EtherCAT_Master_ATxxxx.Beckhoff_AT1xxx.Beckhoff_AT2xxxEK1122.A_0060_AT2020_0250_0019_AT2020_0250.A_0085_AT2050_5500_0018_AT2050_5500.FB_Inputs.Value_Channel[25] <-> FB Inputs/Value Channel 26
//     PlcTask Inputs/GVL_iXlinker.EtherCAT_Master_ATxxxx.Beckhoff_AT1xxx.Beckhoff_AT2xxxEK1122.A_0060_AT2020_0250_0019_AT2020_0250.A_0085_AT2050_5500_0018_AT2050_5500.FB_Inputs.Value_Channel[26] <-> FB Inputs/Value Channel 27
//     PlcTask Inputs/GVL_iXlinker.EtherCAT_Master_ATxxxx.Beckhoff_AT1xxx.Beckhoff_AT2xxxEK1122.A_0060_AT2020_0250_0019_AT2020_0250.A_0085_AT2050_5500_0018_AT2050_5500.FB_Inputs.Value_Channel[27] <-> FB Inputs/Value Channel 28
//     PlcTask Inputs/GVL_iXlinker.EtherCAT_Master_ATxxxx.Beckhoff_AT1xxx.Beckhoff_AT2xxxEK1122.A_0060_AT2020_0250_0019_AT2020_0250.A_0085_AT2050_5500_0018_AT2050_5500.FB_Inputs.Value_Channel[28] <-> FB Inputs/Value Channel 29
//     PlcTask Inputs/GVL_iXlinker.EtherCAT_Master_ATxxxx.Beckhoff_AT1xxx.Beckhoff_AT2xxxEK1122.A_0060_AT2020_0250_0019_AT2020_0250.A_0085_AT2050_5500_0018_AT2050_5500.FB_Inputs.Value_Channel[29] <-> FB Inputs/Value Channel 30
//     PlcTask Inputs/GVL_iXlinker.EtherCAT_Master_ATxxxx.Beckhoff_AT1xxx.Beckhoff_AT2xxxEK1122.A_0060_AT2020_0250_0019_AT2020_0250.A_0085_AT2050_5500_0018_AT2050_5500.FB_Inputs.Value_Channel[30] <-> FB Inputs/Value Channel 31
//     PlcTask Inputs/GVL_iXlinker.EtherCAT_Master_ATxxxx.Beckhoff_AT1xxx.Beckhoff_AT2xxxEK1122.A_0060_AT2020_0250_0019_AT2020_0250.A_0085_AT2050_5500_0018_AT2050_5500.FB_Inputs.Value_Channel[31] <-> FB Inputs/Value Channel 32
//     PlcTask Outputs/GVL_iXlinker.EtherCAT_Master_ATxxxx.Beckhoff_AT1xxx.Beckhoff_AT2xxxEK1122.A_0060_AT2020_0250_0019_AT2020_0250.A_0085_AT2050_5500_0018_AT2050_5500.FB_Outputs.Control <-> FB Outputs/Control
//     PlcTask Inputs/GVL_iXlinker.EtherCAT_Master_ATxxxx.Beckhoff_AT1xxx.Beckhoff_AT2xxxEK1122.A_0060_AT2020_0250_0019_AT2020_0250.A_0085_AT2050_5500_0018_AT2050_5500.WcState.WcState <-> WcState/WcState
//     PlcTask Inputs/GVL_iXlinker.EtherCAT_Master_ATxxxx.Beckhoff_AT1xxx.Beckhoff_AT2xxxEK1122.A_0060_AT2020_0250_0019_AT2020_0250.A_0085_AT2050_5500_0018_AT2050_5500.WcState.InputToggle <-> WcState/InputToggle
//     PlcTask Inputs/GVL_iXlinker.EtherCAT_Master_ATxxxx.Beckhoff_AT1xxx.Beckhoff_AT2xxxEK1122.A_0060_AT2020_0250_0019_AT2020_0250.A_0085_AT2050_5500_0018_AT2050_5500.InfoData.DcOutputShift <-> InfoData/DcOutputShift
//     PlcTask Inputs/GVL_iXlinker.EtherCAT_Master_ATxxxx.Beckhoff_AT1xxx.Beckhoff_AT2xxxEK1122.A_0060_AT2020_0250_0019_AT2020_0250.A_0085_AT2050_5500_0018_AT2050_5500.InfoData.DcInputShift <-> InfoData/DcInputShift
//     PlcTask Inputs/GVL_iXlinker.EtherCAT_Master_ATxxxx.Beckhoff_AT1xxx.Beckhoff_AT2xxxEK1122.A_0060_AT2020_0250_0019_AT2020_0250.A_0085_AT2050_5500_0018_AT2050_5500.InfoData.State <-> InfoData/State
//   PLC/PLC Instance <-> EtherCAT Master ATxxxx/Beckhoff AT1xxx/Beckhoff AT2xxxEK1122/Beckhoff AT2xxxsub EK1100
//     PlcTask Inputs/GVL_iXlinker.EtherCAT_Master_ATxxxx.Beckhoff_AT1xxx.Beckhoff_AT2xxxEK1122.Beckhoff_AT2xxxsub_EK1100.InfoData.State <-> InfoData/State
//   PLC/PLC Instance <-> EtherCAT Master ATxxxx/Beckhoff AT1xxx/Beckhoff AT2xxxEK1122/A_0001(AT2000-0233-0022)
//     PlcTask Inputs/GVL_iXlinker.EtherCAT_Master_ATxxxx.Beckhoff_AT1xxx.Beckhoff_AT2xxxEK1122.A_0001_AT2000_0233_0022.CC_Inputs_14_Ch.Status <-> CC Inputs 14 Ch/Status
//     PlcTask Inputs/GVL_iXlinker.EtherCAT_Master_ATxxxx.Beckhoff_AT1xxx.Beckhoff_AT2xxxEK1122.A_0001_AT2000_0233_0022.CC_Inputs_14_Ch.Current_actual_value_Ch[0] <-> CC Inputs 14 Ch/Current actual value Ch.1
//     PlcTask Inputs/GVL_iXlinker.EtherCAT_Master_ATxxxx.Beckhoff_AT1xxx.Beckhoff_AT2xxxEK1122.A_0001_AT2000_0233_0022.CC_Inputs_14_Ch.Current_actual_value_Ch[1] <-> CC Inputs 14 Ch/Current actual value Ch.2
//     PlcTask Inputs/GVL_iXlinker.EtherCAT_Master_ATxxxx.Beckhoff_AT1xxx.Beckhoff_AT2xxxEK1122.A_0001_AT2000_0233_0022.CC_Inputs_14_Ch.Current_actual_value_Ch[2] <-> CC Inputs 14 Ch/Current actual value Ch.3
//     PlcTask Inputs/GVL_iXlinker.EtherCAT_Master_ATxxxx.Beckhoff_AT1xxx.Beckhoff_AT2xxxEK1122.A_0001_AT2000_0233_0022.CC_Inputs_14_Ch.Current_actual_value_Ch[3] <-> CC Inputs 14 Ch/Current actual value Ch.4
//     PlcTask Inputs/GVL_iXlinker.EtherCAT_Master_ATxxxx.Beckhoff_AT1xxx.Beckhoff_AT2xxxEK1122.A_0001_AT2000_0233_0022.CC_Inputs_14_Ch.Current_actual_value_Ch[4] <-> CC Inputs 14 Ch/Current actual value Ch.5
//     PlcTask Inputs/GVL_iXlinker.EtherCAT_Master_ATxxxx.Beckhoff_AT1xxx.Beckhoff_AT2xxxEK1122.A_0001_AT2000_0233_0022.CC_Inputs_14_Ch.Current_actual_value_Ch[5] <-> CC Inputs 14 Ch/Current actual value Ch.6
//     PlcTask Inputs/GVL_iXlinker.EtherCAT_Master_ATxxxx.Beckhoff_AT1xxx.Beckhoff_AT2xxxEK1122.A_0001_AT2000_0233_0022.CC_Inputs_14_Ch.Current_actual_value_Ch[6] <-> CC Inputs 14 Ch/Current actual value Ch.7
//     PlcTask Inputs/GVL_iXlinker.EtherCAT_Master_ATxxxx.Beckhoff_AT1xxx.Beckhoff_AT2xxxEK1122.A_0001_AT2000_0233_0022.CC_Inputs_14_Ch.Current_actual_value_Ch[7] <-> CC Inputs 14 Ch/Current actual value Ch.8
//     PlcTask Inputs/GVL_iXlinker.EtherCAT_Master_ATxxxx.Beckhoff_AT1xxx.Beckhoff_AT2xxxEK1122.A_0001_AT2000_0233_0022.CC_Inputs_14_Ch.Current_actual_value_Ch[8] <-> CC Inputs 14 Ch/Current actual value Ch.9
//     PlcTask Inputs/GVL_iXlinker.EtherCAT_Master_ATxxxx.Beckhoff_AT1xxx.Beckhoff_AT2xxxEK1122.A_0001_AT2000_0233_0022.CC_Inputs_14_Ch.Current_actual_value_Ch[9] <-> CC Inputs 14 Ch/Current actual value Ch.10
//     PlcTask Inputs/GVL_iXlinker.EtherCAT_Master_ATxxxx.Beckhoff_AT1xxx.Beckhoff_AT2xxxEK1122.A_0001_AT2000_0233_0022.CC_Inputs_14_Ch.Current_actual_value_Ch[10] <-> CC Inputs 14 Ch/Current actual value Ch.11
//     PlcTask Inputs/GVL_iXlinker.EtherCAT_Master_ATxxxx.Beckhoff_AT1xxx.Beckhoff_AT2xxxEK1122.A_0001_AT2000_0233_0022.CC_Inputs_14_Ch.Current_actual_value_Ch[11] <-> CC Inputs 14 Ch/Current actual value Ch.12
//     PlcTask Inputs/GVL_iXlinker.EtherCAT_Master_ATxxxx.Beckhoff_AT1xxx.Beckhoff_AT2xxxEK1122.A_0001_AT2000_0233_0022.CC_Inputs_14_Ch.Current_actual_value_Ch[12] <-> CC Inputs 14 Ch/Current actual value Ch.13
//     PlcTask Inputs/GVL_iXlinker.EtherCAT_Master_ATxxxx.Beckhoff_AT1xxx.Beckhoff_AT2xxxEK1122.A_0001_AT2000_0233_0022.CC_Inputs_14_Ch.Current_actual_value_Ch[13] <-> CC Inputs 14 Ch/Current actual value Ch.14
//     PlcTask Outputs/GVL_iXlinker.EtherCAT_Master_ATxxxx.Beckhoff_AT1xxx.Beckhoff_AT2xxxEK1122.A_0001_AT2000_0233_0022.CC_Outputs_14_Ch.Control <-> CC Outputs 14 Ch/Control
//     PlcTask Outputs/GVL_iXlinker.EtherCAT_Master_ATxxxx.Beckhoff_AT1xxx.Beckhoff_AT2xxxEK1122.A_0001_AT2000_0233_0022.CC_Outputs_14_Ch.Current_setpoint_value_Ch[0] <-> CC Outputs 14 Ch/Current setpoint value Ch.1
//     PlcTask Outputs/GVL_iXlinker.EtherCAT_Master_ATxxxx.Beckhoff_AT1xxx.Beckhoff_AT2xxxEK1122.A_0001_AT2000_0233_0022.CC_Outputs_14_Ch.Current_setpoint_value_Ch[1] <-> CC Outputs 14 Ch/Current setpoint value Ch.2
//     PlcTask Outputs/GVL_iXlinker.EtherCAT_Master_ATxxxx.Beckhoff_AT1xxx.Beckhoff_AT2xxxEK1122.A_0001_AT2000_0233_0022.CC_Outputs_14_Ch.Current_setpoint_value_Ch[2] <-> CC Outputs 14 Ch/Current setpoint value Ch.3
//     PlcTask Outputs/GVL_iXlinker.EtherCAT_Master_ATxxxx.Beckhoff_AT1xxx.Beckhoff_AT2xxxEK1122.A_0001_AT2000_0233_0022.CC_Outputs_14_Ch.Current_setpoint_value_Ch[3] <-> CC Outputs 14 Ch/Current setpoint value Ch.4
//     PlcTask Outputs/GVL_iXlinker.EtherCAT_Master_ATxxxx.Beckhoff_AT1xxx.Beckhoff_AT2xxxEK1122.A_0001_AT2000_0233_0022.CC_Outputs_14_Ch.Current_setpoint_value_Ch[4] <-> CC Outputs 14 Ch/Current setpoint value Ch.5
//     PlcTask Outputs/GVL_iXlinker.EtherCAT_Master_ATxxxx.Beckhoff_AT1xxx.Beckhoff_AT2xxxEK1122.A_0001_AT2000_0233_0022.CC_Outputs_14_Ch.Current_setpoint_value_Ch[5] <-> CC Outputs 14 Ch/Current setpoint value Ch.6
//     PlcTask Outputs/GVL_iXlinker.EtherCAT_Master_ATxxxx.Beckhoff_AT1xxx.Beckhoff_AT2xxxEK1122.A_0001_AT2000_0233_0022.CC_Outputs_14_Ch.Current_setpoint_value_Ch[6] <-> CC Outputs 14 Ch/Current setpoint value Ch.7
//     PlcTask Outputs/GVL_iXlinker.EtherCAT_Master_ATxxxx.Beckhoff_AT1xxx.Beckhoff_AT2xxxEK1122.A_0001_AT2000_0233_0022.CC_Outputs_14_Ch.Current_setpoint_value_Ch[7] <-> CC Outputs 14 Ch/Current setpoint value Ch.8
//     PlcTask Outputs/GVL_iXlinker.EtherCAT_Master_ATxxxx.Beckhoff_AT1xxx.Beckhoff_AT2xxxEK1122.A_0001_AT2000_0233_0022.CC_Outputs_14_Ch.Current_setpoint_value_Ch[8] <-> CC Outputs 14 Ch/Current setpoint value Ch.9
//     PlcTask Outputs/GVL_iXlinker.EtherCAT_Master_ATxxxx.Beckhoff_AT1xxx.Beckhoff_AT2xxxEK1122.A_0001_AT2000_0233_0022.CC_Outputs_14_Ch.Current_setpoint_value_Ch[9] <-> CC Outputs 14 Ch/Current setpoint value Ch.10
//     PlcTask Outputs/GVL_iXlinker.EtherCAT_Master_ATxxxx.Beckhoff_AT1xxx.Beckhoff_AT2xxxEK1122.A_0001_AT2000_0233_0022.CC_Outputs_14_Ch.Current_setpoint_value_Ch[10] <-> CC Outputs 14 Ch/Current setpoint value Ch.11
//     PlcTask Outputs/GVL_iXlinker.EtherCAT_Master_ATxxxx.Beckhoff_AT1xxx.Beckhoff_AT2xxxEK1122.A_0001_AT2000_0233_0022.CC_Outputs_14_Ch.Current_setpoint_value_Ch[11] <-> CC Outputs 14 Ch/Current setpoint value Ch.12
//     PlcTask Outputs/GVL_iXlinker.EtherCAT_Master_ATxxxx.Beckhoff_AT1xxx.Beckhoff_AT2xxxEK1122.A_0001_AT2000_0233_0022.CC_Outputs_14_Ch.Current_setpoint_value_Ch[12] <-> CC Outputs 14 Ch/Current setpoint value Ch.13
//     PlcTask Outputs/GVL_iXlinker.EtherCAT_Master_ATxxxx.Beckhoff_AT1xxx.Beckhoff_AT2xxxEK1122.A_0001_AT2000_0233_0022.CC_Outputs_14_Ch.Current_setpoint_value_Ch[13] <-> CC Outputs 14 Ch/Current setpoint value Ch.14
//     PlcTask Inputs/GVL_iXlinker.EtherCAT_Master_ATxxxx.Beckhoff_AT1xxx.Beckhoff_AT2xxxEK1122.A_0001_AT2000_0233_0022.WcState.WcState <-> WcState/WcState
//     PlcTask Inputs/GVL_iXlinker.EtherCAT_Master_ATxxxx.Beckhoff_AT1xxx.Beckhoff_AT2xxxEK1122.A_0001_AT2000_0233_0022.WcState.InputToggle <-> WcState/InputToggle
//     PlcTask Inputs/GVL_iXlinker.EtherCAT_Master_ATxxxx.Beckhoff_AT1xxx.Beckhoff_AT2xxxEK1122.A_0001_AT2000_0233_0022.InfoData.AdsAddr <-> InfoData/AdsAddr
//     PlcTask Inputs/GVL_iXlinker.EtherCAT_Master_ATxxxx.Beckhoff_AT1xxx.Beckhoff_AT2xxxEK1122.A_0001_AT2000_0233_0022.InfoData.DcOutputShift <-> InfoData/DcOutputShift
//     PlcTask Inputs/GVL_iXlinker.EtherCAT_Master_ATxxxx.Beckhoff_AT1xxx.Beckhoff_AT2xxxEK1122.A_0001_AT2000_0233_0022.InfoData.DcInputShift <-> InfoData/DcInputShift
//     PlcTask Inputs/GVL_iXlinker.EtherCAT_Master_ATxxxx.Beckhoff_AT1xxx.Beckhoff_AT2xxxEK1122.A_0001_AT2000_0233_0022.InfoData.State <-> InfoData/State
//   PLC/PLC Instance <-> EtherCAT Master ATxxxx/Beckhoff AT1xxx/Beckhoff AT2xxxEK1122/A_0002(AT2000-0233-0023)
//     PlcTask Inputs/GVL_iXlinker.EtherCAT_Master_ATxxxx.Beckhoff_AT1xxx.Beckhoff_AT2xxxEK1122.A_0002_AT2000_0233_0023.CC_Inputs_14_Ch.Status <-> CC Inputs 14 Ch/Status
//     PlcTask Inputs/GVL_iXlinker.EtherCAT_Master_ATxxxx.Beckhoff_AT1xxx.Beckhoff_AT2xxxEK1122.A_0002_AT2000_0233_0023.CC_Inputs_14_Ch.Current_actual_value_Ch[0] <-> CC Inputs 14 Ch/Current actual value Ch.1
//     PlcTask Inputs/GVL_iXlinker.EtherCAT_Master_ATxxxx.Beckhoff_AT1xxx.Beckhoff_AT2xxxEK1122.A_0002_AT2000_0233_0023.CC_Inputs_14_Ch.Current_actual_value_Ch[1] <-> CC Inputs 14 Ch/Current actual value Ch.2
//     PlcTask Inputs/GVL_iXlinker.EtherCAT_Master_ATxxxx.Beckhoff_AT1xxx.Beckhoff_AT2xxxEK1122.A_0002_AT2000_0233_0023.CC_Inputs_14_Ch.Current_actual_value_Ch[2] <-> CC Inputs 14 Ch/Current actual value Ch.3
//     PlcTask Inputs/GVL_iXlinker.EtherCAT_Master_ATxxxx.Beckhoff_AT1xxx.Beckhoff_AT2xxxEK1122.A_0002_AT2000_0233_0023.CC_Inputs_14_Ch.Current_actual_value_Ch[3] <-> CC Inputs 14 Ch/Current actual value Ch.4
//     PlcTask Inputs/GVL_iXlinker.EtherCAT_Master_ATxxxx.Beckhoff_AT1xxx.Beckhoff_AT2xxxEK1122.A_0002_AT2000_0233_0023.CC_Inputs_14_Ch.Current_actual_value_Ch[4] <-> CC Inputs 14 Ch/Current actual value Ch.5
//     PlcTask Inputs/GVL_iXlinker.EtherCAT_Master_ATxxxx.Beckhoff_AT1xxx.Beckhoff_AT2xxxEK1122.A_0002_AT2000_0233_0023.CC_Inputs_14_Ch.Current_actual_value_Ch[5] <-> CC Inputs 14 Ch/Current actual value Ch.6
//     PlcTask Inputs/GVL_iXlinker.EtherCAT_Master_ATxxxx.Beckhoff_AT1xxx.Beckhoff_AT2xxxEK1122.A_0002_AT2000_0233_0023.CC_Inputs_14_Ch.Current_actual_value_Ch[6] <-> CC Inputs 14 Ch/Current actual value Ch.7
//     PlcTask Inputs/GVL_iXlinker.EtherCAT_Master_ATxxxx.Beckhoff_AT1xxx.Beckhoff_AT2xxxEK1122.A_0002_AT2000_0233_0023.CC_Inputs_14_Ch.Current_actual_value_Ch[7] <-> CC Inputs 14 Ch/Current actual value Ch.8
//     PlcTask Inputs/GVL_iXlinker.EtherCAT_Master_ATxxxx.Beckhoff_AT1xxx.Beckhoff_AT2xxxEK1122.A_0002_AT2000_0233_0023.CC_Inputs_14_Ch.Current_actual_value_Ch[8] <-> CC Inputs 14 Ch/Current actual value Ch.9
//     PlcTask Inputs/GVL_iXlinker.EtherCAT_Master_ATxxxx.Beckhoff_AT1xxx.Beckhoff_AT2xxxEK1122.A_0002_AT2000_0233_0023.CC_Inputs_14_Ch.Current_actual_value_Ch[9] <-> CC Inputs 14 Ch/Current actual value Ch.10
//     PlcTask Inputs/GVL_iXlinker.EtherCAT_Master_ATxxxx.Beckhoff_AT1xxx.Beckhoff_AT2xxxEK1122.A_0002_AT2000_0233_0023.CC_Inputs_14_Ch.Current_actual_value_Ch[10] <-> CC Inputs 14 Ch/Current actual value Ch.11
//     PlcTask Inputs/GVL_iXlinker.EtherCAT_Master_ATxxxx.Beckhoff_AT1xxx.Beckhoff_AT2xxxEK1122.A_0002_AT2000_0233_0023.CC_Inputs_14_Ch.Current_actual_value_Ch[11] <-> CC Inputs 14 Ch/Current actual value Ch.12
//     PlcTask Inputs/GVL_iXlinker.EtherCAT_Master_ATxxxx.Beckhoff_AT1xxx.Beckhoff_AT2xxxEK1122.A_0002_AT2000_0233_0023.CC_Inputs_14_Ch.Current_actual_value_Ch[12] <-> CC Inputs 14 Ch/Current actual value Ch.13
//     PlcTask Inputs/GVL_iXlinker.EtherCAT_Master_ATxxxx.Beckhoff_AT1xxx.Beckhoff_AT2xxxEK1122.A_0002_AT2000_0233_0023.CC_Inputs_14_Ch.Current_actual_value_Ch[13] <-> CC Inputs 14 Ch/Current actual value Ch.14
//     PlcTask Outputs/GVL_iXlinker.EtherCAT_Master_ATxxxx.Beckhoff_AT1xxx.Beckhoff_AT2xxxEK1122.A_0002_AT2000_0233_0023.CC_Outputs_14_Ch.Control <-> CC Outputs 14 Ch/Control
//     PlcTask Outputs/GVL_iXlinker.EtherCAT_Master_ATxxxx.Beckhoff_AT1xxx.Beckhoff_AT2xxxEK1122.A_0002_AT2000_0233_0023.CC_Outputs_14_Ch.Current_setpoint_value_Ch[0] <-> CC Outputs 14 Ch/Current setpoint value Ch.1
//     PlcTask Outputs/GVL_iXlinker.EtherCAT_Master_ATxxxx.Beckhoff_AT1xxx.Beckhoff_AT2xxxEK1122.A_0002_AT2000_0233_0023.CC_Outputs_14_Ch.Current_setpoint_value_Ch[1] <-> CC Outputs 14 Ch/Current setpoint value Ch.2
//     PlcTask Outputs/GVL_iXlinker.EtherCAT_Master_ATxxxx.Beckhoff_AT1xxx.Beckhoff_AT2xxxEK1122.A_0002_AT2000_0233_0023.CC_Outputs_14_Ch.Current_setpoint_value_Ch[2] <-> CC Outputs 14 Ch/Current setpoint value Ch.3
//     PlcTask Outputs/GVL_iXlinker.EtherCAT_Master_ATxxxx.Beckhoff_AT1xxx.Beckhoff_AT2xxxEK1122.A_0002_AT2000_0233_0023.CC_Outputs_14_Ch.Current_setpoint_value_Ch[3] <-> CC Outputs 14 Ch/Current setpoint value Ch.4
//     PlcTask Outputs/GVL_iXlinker.EtherCAT_Master_ATxxxx.Beckhoff_AT1xxx.Beckhoff_AT2xxxEK1122.A_0002_AT2000_0233_0023.CC_Outputs_14_Ch.Current_setpoint_value_Ch[4] <-> CC Outputs 14 Ch/Current setpoint value Ch.5
//     PlcTask Outputs/GVL_iXlinker.EtherCAT_Master_ATxxxx.Beckhoff_AT1xxx.Beckhoff_AT2xxxEK1122.A_0002_AT2000_0233_0023.CC_Outputs_14_Ch.Current_setpoint_value_Ch[5] <-> CC Outputs 14 Ch/Current setpoint value Ch.6
//     PlcTask Outputs/GVL_iXlinker.EtherCAT_Master_ATxxxx.Beckhoff_AT1xxx.Beckhoff_AT2xxxEK1122.A_0002_AT2000_0233_0023.CC_Outputs_14_Ch.Current_setpoint_value_Ch[6] <-> CC Outputs 14 Ch/Current setpoint value Ch.7
//     PlcTask Outputs/GVL_iXlinker.EtherCAT_Master_ATxxxx.Beckhoff_AT1xxx.Beckhoff_AT2xxxEK1122.A_0002_AT2000_0233_0023.CC_Outputs_14_Ch.Current_setpoint_value_Ch[7] <-> CC Outputs 14 Ch/Current setpoint value Ch.8
//     PlcTask Outputs/GVL_iXlinker.EtherCAT_Master_ATxxxx.Beckhoff_AT1xxx.Beckhoff_AT2xxxEK1122.A_0002_AT2000_0233_0023.CC_Outputs_14_Ch.Current_setpoint_value_Ch[8] <-> CC Outputs 14 Ch/Current setpoint value Ch.9
//     PlcTask Outputs/GVL_iXlinker.EtherCAT_Master_ATxxxx.Beckhoff_AT1xxx.Beckhoff_AT2xxxEK1122.A_0002_AT2000_0233_0023.CC_Outputs_14_Ch.Current_setpoint_value_Ch[9] <-> CC Outputs 14 Ch/Current setpoint value Ch.10
//     PlcTask Outputs/GVL_iXlinker.EtherCAT_Master_ATxxxx.Beckhoff_AT1xxx.Beckhoff_AT2xxxEK1122.A_0002_AT2000_0233_0023.CC_Outputs_14_Ch.Current_setpoint_value_Ch[10] <-> CC Outputs 14 Ch/Current setpoint value Ch.11
//     PlcTask Outputs/GVL_iXlinker.EtherCAT_Master_ATxxxx.Beckhoff_AT1xxx.Beckhoff_AT2xxxEK1122.A_0002_AT2000_0233_0023.CC_Outputs_14_Ch.Current_setpoint_value_Ch[11] <-> CC Outputs 14 Ch/Current setpoint value Ch.12
//     PlcTask Outputs/GVL_iXlinker.EtherCAT_Master_ATxxxx.Beckhoff_AT1xxx.Beckhoff_AT2xxxEK1122.A_0002_AT2000_0233_0023.CC_Outputs_14_Ch.Current_setpoint_value_Ch[12] <-> CC Outputs 14 Ch/Current setpoint value Ch.13
//     PlcTask Outputs/GVL_iXlinker.EtherCAT_Master_ATxxxx.Beckhoff_AT1xxx.Beckhoff_AT2xxxEK1122.A_0002_AT2000_0233_0023.CC_Outputs_14_Ch.Current_setpoint_value_Ch[13] <-> CC Outputs 14 Ch/Current setpoint value Ch.14
//     PlcTask Inputs/GVL_iXlinker.EtherCAT_Master_ATxxxx.Beckhoff_AT1xxx.Beckhoff_AT2xxxEK1122.A_0002_AT2000_0233_0023.WcState.WcState <-> WcState/WcState
//     PlcTask Inputs/GVL_iXlinker.EtherCAT_Master_ATxxxx.Beckhoff_AT1xxx.Beckhoff_AT2xxxEK1122.A_0002_AT2000_0233_0023.WcState.InputToggle <-> WcState/InputToggle
//     PlcTask Inputs/GVL_iXlinker.EtherCAT_Master_ATxxxx.Beckhoff_AT1xxx.Beckhoff_AT2xxxEK1122.A_0002_AT2000_0233_0023.InfoData.AdsAddr <-> InfoData/AdsAddr
//     PlcTask Inputs/GVL_iXlinker.EtherCAT_Master_ATxxxx.Beckhoff_AT1xxx.Beckhoff_AT2xxxEK1122.A_0002_AT2000_0233_0023.InfoData.DcOutputShift <-> InfoData/DcOutputShift
//     PlcTask Inputs/GVL_iXlinker.EtherCAT_Master_ATxxxx.Beckhoff_AT1xxx.Beckhoff_AT2xxxEK1122.A_0002_AT2000_0233_0023.InfoData.DcInputShift <-> InfoData/DcInputShift
//     PlcTask Inputs/GVL_iXlinker.EtherCAT_Master_ATxxxx.Beckhoff_AT1xxx.Beckhoff_AT2xxxEK1122.A_0002_AT2000_0233_0023.InfoData.State <-> InfoData/State
//   PLC/PLC Instance <-> EtherCAT Master ATxxxx/Beckhoff AT1xxx/Beckhoff AT2xxxEK1122/A_0003(AT2000-0233-0024)
//     PlcTask Inputs/GVL_iXlinker.EtherCAT_Master_ATxxxx.Beckhoff_AT1xxx.Beckhoff_AT2xxxEK1122.A_0003_AT2000_0233_0024.CC_Inputs_14_Ch.Status <-> CC Inputs 14 Ch/Status
//     PlcTask Inputs/GVL_iXlinker.EtherCAT_Master_ATxxxx.Beckhoff_AT1xxx.Beckhoff_AT2xxxEK1122.A_0003_AT2000_0233_0024.CC_Inputs_14_Ch.Current_actual_value_Ch[0] <-> CC Inputs 14 Ch/Current actual value Ch.1
//     PlcTask Inputs/GVL_iXlinker.EtherCAT_Master_ATxxxx.Beckhoff_AT1xxx.Beckhoff_AT2xxxEK1122.A_0003_AT2000_0233_0024.CC_Inputs_14_Ch.Current_actual_value_Ch[1] <-> CC Inputs 14 Ch/Current actual value Ch.2
//     PlcTask Inputs/GVL_iXlinker.EtherCAT_Master_ATxxxx.Beckhoff_AT1xxx.Beckhoff_AT2xxxEK1122.A_0003_AT2000_0233_0024.CC_Inputs_14_Ch.Current_actual_value_Ch[2] <-> CC Inputs 14 Ch/Current actual value Ch.3
//     PlcTask Inputs/GVL_iXlinker.EtherCAT_Master_ATxxxx.Beckhoff_AT1xxx.Beckhoff_AT2xxxEK1122.A_0003_AT2000_0233_0024.CC_Inputs_14_Ch.Current_actual_value_Ch[3] <-> CC Inputs 14 Ch/Current actual value Ch.4
//     PlcTask Inputs/GVL_iXlinker.EtherCAT_Master_ATxxxx.Beckhoff_AT1xxx.Beckhoff_AT2xxxEK1122.A_0003_AT2000_0233_0024.CC_Inputs_14_Ch.Current_actual_value_Ch[4] <-> CC Inputs 14 Ch/Current actual value Ch.5
//     PlcTask Inputs/GVL_iXlinker.EtherCAT_Master_ATxxxx.Beckhoff_AT1xxx.Beckhoff_AT2xxxEK1122.A_0003_AT2000_0233_0024.CC_Inputs_14_Ch.Current_actual_value_Ch[5] <-> CC Inputs 14 Ch/Current actual value Ch.6
//     PlcTask Inputs/GVL_iXlinker.EtherCAT_Master_ATxxxx.Beckhoff_AT1xxx.Beckhoff_AT2xxxEK1122.A_0003_AT2000_0233_0024.CC_Inputs_14_Ch.Current_actual_value_Ch[6] <-> CC Inputs 14 Ch/Current actual value Ch.7
//     PlcTask Inputs/GVL_iXlinker.EtherCAT_Master_ATxxxx.Beckhoff_AT1xxx.Beckhoff_AT2xxxEK1122.A_0003_AT2000_0233_0024.CC_Inputs_14_Ch.Current_actual_value_Ch[7] <-> CC Inputs 14 Ch/Current actual value Ch.8
//     PlcTask Inputs/GVL_iXlinker.EtherCAT_Master_ATxxxx.Beckhoff_AT1xxx.Beckhoff_AT2xxxEK1122.A_0003_AT2000_0233_0024.CC_Inputs_14_Ch.Current_actual_value_Ch[8] <-> CC Inputs 14 Ch/Current actual value Ch.9
//     PlcTask Inputs/GVL_iXlinker.EtherCAT_Master_ATxxxx.Beckhoff_AT1xxx.Beckhoff_AT2xxxEK1122.A_0003_AT2000_0233_0024.CC_Inputs_14_Ch.Current_actual_value_Ch[9] <-> CC Inputs 14 Ch/Current actual value Ch.10
//     PlcTask Inputs/GVL_iXlinker.EtherCAT_Master_ATxxxx.Beckhoff_AT1xxx.Beckhoff_AT2xxxEK1122.A_0003_AT2000_0233_0024.CC_Inputs_14_Ch.Current_actual_value_Ch[10] <-> CC Inputs 14 Ch/Current actual value Ch.11
//     PlcTask Inputs/GVL_iXlinker.EtherCAT_Master_ATxxxx.Beckhoff_AT1xxx.Beckhoff_AT2xxxEK1122.A_0003_AT2000_0233_0024.CC_Inputs_14_Ch.Current_actual_value_Ch[11] <-> CC Inputs 14 Ch/Current actual value Ch.12
//     PlcTask Inputs/GVL_iXlinker.EtherCAT_Master_ATxxxx.Beckhoff_AT1xxx.Beckhoff_AT2xxxEK1122.A_0003_AT2000_0233_0024.CC_Inputs_14_Ch.Current_actual_value_Ch[12] <-> CC Inputs 14 Ch/Current actual value Ch.13
//     PlcTask Inputs/GVL_iXlinker.EtherCAT_Master_ATxxxx.Beckhoff_AT1xxx.Beckhoff_AT2xxxEK1122.A_0003_AT2000_0233_0024.CC_Inputs_14_Ch.Current_actual_value_Ch[13] <-> CC Inputs 14 Ch/Current actual value Ch.14
//     PlcTask Outputs/GVL_iXlinker.EtherCAT_Master_ATxxxx.Beckhoff_AT1xxx.Beckhoff_AT2xxxEK1122.A_0003_AT2000_0233_0024.CC_Outputs_14_Ch.Control <-> CC Outputs 14 Ch/Control
//     PlcTask Outputs/GVL_iXlinker.EtherCAT_Master_ATxxxx.Beckhoff_AT1xxx.Beckhoff_AT2xxxEK1122.A_0003_AT2000_0233_0024.CC_Outputs_14_Ch.Current_setpoint_value_Ch[0] <-> CC Outputs 14 Ch/Current setpoint value Ch.1
//     PlcTask Outputs/GVL_iXlinker.EtherCAT_Master_ATxxxx.Beckhoff_AT1xxx.Beckhoff_AT2xxxEK1122.A_0003_AT2000_0233_0024.CC_Outputs_14_Ch.Current_setpoint_value_Ch[1] <-> CC Outputs 14 Ch/Current setpoint value Ch.2
//     PlcTask Outputs/GVL_iXlinker.EtherCAT_Master_ATxxxx.Beckhoff_AT1xxx.Beckhoff_AT2xxxEK1122.A_0003_AT2000_0233_0024.CC_Outputs_14_Ch.Current_setpoint_value_Ch[2] <-> CC Outputs 14 Ch/Current setpoint value Ch.3
//     PlcTask Outputs/GVL_iXlinker.EtherCAT_Master_ATxxxx.Beckhoff_AT1xxx.Beckhoff_AT2xxxEK1122.A_0003_AT2000_0233_0024.CC_Outputs_14_Ch.Current_setpoint_value_Ch[3] <-> CC Outputs 14 Ch/Current setpoint value Ch.4
//     PlcTask Outputs/GVL_iXlinker.EtherCAT_Master_ATxxxx.Beckhoff_AT1xxx.Beckhoff_AT2xxxEK1122.A_0003_AT2000_0233_0024.CC_Outputs_14_Ch.Current_setpoint_value_Ch[4] <-> CC Outputs 14 Ch/Current setpoint value Ch.5
//     PlcTask Outputs/GVL_iXlinker.EtherCAT_Master_ATxxxx.Beckhoff_AT1xxx.Beckhoff_AT2xxxEK1122.A_0003_AT2000_0233_0024.CC_Outputs_14_Ch.Current_setpoint_value_Ch[5] <-> CC Outputs 14 Ch/Current setpoint value Ch.6
//     PlcTask Outputs/GVL_iXlinker.EtherCAT_Master_ATxxxx.Beckhoff_AT1xxx.Beckhoff_AT2xxxEK1122.A_0003_AT2000_0233_0024.CC_Outputs_14_Ch.Current_setpoint_value_Ch[6] <-> CC Outputs 14 Ch/Current setpoint value Ch.7
//     PlcTask Outputs/GVL_iXlinker.EtherCAT_Master_ATxxxx.Beckhoff_AT1xxx.Beckhoff_AT2xxxEK1122.A_0003_AT2000_0233_0024.CC_Outputs_14_Ch.Current_setpoint_value_Ch[7] <-> CC Outputs 14 Ch/Current setpoint value Ch.8
//     PlcTask Outputs/GVL_iXlinker.EtherCAT_Master_ATxxxx.Beckhoff_AT1xxx.Beckhoff_AT2xxxEK1122.A_0003_AT2000_0233_0024.CC_Outputs_14_Ch.Current_setpoint_value_Ch[8] <-> CC Outputs 14 Ch/Current setpoint value Ch.9
//     PlcTask Outputs/GVL_iXlinker.EtherCAT_Master_ATxxxx.Beckhoff_AT1xxx.Beckhoff_AT2xxxEK1122.A_0003_AT2000_0233_0024.CC_Outputs_14_Ch.Current_setpoint_value_Ch[9] <-> CC Outputs 14 Ch/Current setpoint value Ch.10
//     PlcTask Outputs/GVL_iXlinker.EtherCAT_Master_ATxxxx.Beckhoff_AT1xxx.Beckhoff_AT2xxxEK1122.A_0003_AT2000_0233_0024.CC_Outputs_14_Ch.Current_setpoint_value_Ch[10] <-> CC Outputs 14 Ch/Current setpoint value Ch.11
//     PlcTask Outputs/GVL_iXlinker.EtherCAT_Master_ATxxxx.Beckhoff_AT1xxx.Beckhoff_AT2xxxEK1122.A_0003_AT2000_0233_0024.CC_Outputs_14_Ch.Current_setpoint_value_Ch[11] <-> CC Outputs 14 Ch/Current setpoint value Ch.12
//     PlcTask Outputs/GVL_iXlinker.EtherCAT_Master_ATxxxx.Beckhoff_AT1xxx.Beckhoff_AT2xxxEK1122.A_0003_AT2000_0233_0024.CC_Outputs_14_Ch.Current_setpoint_value_Ch[12] <-> CC Outputs 14 Ch/Current setpoint value Ch.13
//     PlcTask Outputs/GVL_iXlinker.EtherCAT_Master_ATxxxx.Beckhoff_AT1xxx.Beckhoff_AT2xxxEK1122.A_0003_AT2000_0233_0024.CC_Outputs_14_Ch.Current_setpoint_value_Ch[13] <-> CC Outputs 14 Ch/Current setpoint value Ch.14
//     PlcTask Inputs/GVL_iXlinker.EtherCAT_Master_ATxxxx.Beckhoff_AT1xxx.Beckhoff_AT2xxxEK1122.A_0003_AT2000_0233_0024.WcState.WcState <-> WcState/WcState
//     PlcTask Inputs/GVL_iXlinker.EtherCAT_Master_ATxxxx.Beckhoff_AT1xxx.Beckhoff_AT2xxxEK1122.A_0003_AT2000_0233_0024.WcState.InputToggle <-> WcState/InputToggle
//     PlcTask Inputs/GVL_iXlinker.EtherCAT_Master_ATxxxx.Beckhoff_AT1xxx.Beckhoff_AT2xxxEK1122.A_0003_AT2000_0233_0024.InfoData.AdsAddr <-> InfoData/AdsAddr
//     PlcTask Inputs/GVL_iXlinker.EtherCAT_Master_ATxxxx.Beckhoff_AT1xxx.Beckhoff_AT2xxxEK1122.A_0003_AT2000_0233_0024.InfoData.DcOutputShift <-> InfoData/DcOutputShift
//     PlcTask Inputs/GVL_iXlinker.EtherCAT_Master_ATxxxx.Beckhoff_AT1xxx.Beckhoff_AT2xxxEK1122.A_0003_AT2000_0233_0024.InfoData.DcInputShift <-> InfoData/DcInputShift
//     PlcTask Inputs/GVL_iXlinker.EtherCAT_Master_ATxxxx.Beckhoff_AT1xxx.Beckhoff_AT2xxxEK1122.A_0003_AT2000_0233_0024.InfoData.State <-> InfoData/State
//   PLC/PLC Instance <-> EtherCAT Master ATxxxx/Beckhoff AT1xxx/Beckhoff AT2xxxEK1122/A_0004(AT2000-0250-0016)
//     PlcTask Inputs/GVL_iXlinker.EtherCAT_Master_ATxxxx.Beckhoff_AT1xxx.Beckhoff_AT2xxxEK1122.A_0004_AT2000_0250_0016.CC_Inputs.Status <-> CC Inputs/Status
//     PlcTask Inputs/GVL_iXlinker.EtherCAT_Master_ATxxxx.Beckhoff_AT1xxx.Beckhoff_AT2xxxEK1122.A_0004_AT2000_0250_0016.CC_Inputs.Current_actual_value_Ch[0] <-> CC Inputs/Current actual value Ch.1
//     PlcTask Inputs/GVL_iXlinker.EtherCAT_Master_ATxxxx.Beckhoff_AT1xxx.Beckhoff_AT2xxxEK1122.A_0004_AT2000_0250_0016.CC_Inputs.Current_actual_value_Ch[1] <-> CC Inputs/Current actual value Ch.2
//     PlcTask Inputs/GVL_iXlinker.EtherCAT_Master_ATxxxx.Beckhoff_AT1xxx.Beckhoff_AT2xxxEK1122.A_0004_AT2000_0250_0016.CC_Inputs.Current_actual_value_Ch[2] <-> CC Inputs/Current actual value Ch.3
//     PlcTask Inputs/GVL_iXlinker.EtherCAT_Master_ATxxxx.Beckhoff_AT1xxx.Beckhoff_AT2xxxEK1122.A_0004_AT2000_0250_0016.CC_Inputs.Current_actual_value_Ch[3] <-> CC Inputs/Current actual value Ch.4
//     PlcTask Inputs/GVL_iXlinker.EtherCAT_Master_ATxxxx.Beckhoff_AT1xxx.Beckhoff_AT2xxxEK1122.A_0004_AT2000_0250_0016.CC_Inputs.Current_actual_value_Ch[4] <-> CC Inputs/Current actual value Ch.5
//     PlcTask Inputs/GVL_iXlinker.EtherCAT_Master_ATxxxx.Beckhoff_AT1xxx.Beckhoff_AT2xxxEK1122.A_0004_AT2000_0250_0016.CC_Inputs.Current_actual_value_Ch[5] <-> CC Inputs/Current actual value Ch.6
//     PlcTask Inputs/GVL_iXlinker.EtherCAT_Master_ATxxxx.Beckhoff_AT1xxx.Beckhoff_AT2xxxEK1122.A_0004_AT2000_0250_0016.CC_Inputs.Current_actual_value_Ch[6] <-> CC Inputs/Current actual value Ch.7
//     PlcTask Inputs/GVL_iXlinker.EtherCAT_Master_ATxxxx.Beckhoff_AT1xxx.Beckhoff_AT2xxxEK1122.A_0004_AT2000_0250_0016.CC_Inputs.Current_actual_value_Ch[7] <-> CC Inputs/Current actual value Ch.8
//     PlcTask Inputs/GVL_iXlinker.EtherCAT_Master_ATxxxx.Beckhoff_AT1xxx.Beckhoff_AT2xxxEK1122.A_0004_AT2000_0250_0016.CC_Inputs.Current_actual_value_Ch[8] <-> CC Inputs/Current actual value Ch.9
//     PlcTask Inputs/GVL_iXlinker.EtherCAT_Master_ATxxxx.Beckhoff_AT1xxx.Beckhoff_AT2xxxEK1122.A_0004_AT2000_0250_0016.CC_Inputs.Current_actual_value_Ch[9] <-> CC Inputs/Current actual value Ch.10
//     PlcTask Inputs/GVL_iXlinker.EtherCAT_Master_ATxxxx.Beckhoff_AT1xxx.Beckhoff_AT2xxxEK1122.A_0004_AT2000_0250_0016.CC_Inputs.Current_actual_value_Ch[10] <-> CC Inputs/Current actual value Ch.11
//     PlcTask Inputs/GVL_iXlinker.EtherCAT_Master_ATxxxx.Beckhoff_AT1xxx.Beckhoff_AT2xxxEK1122.A_0004_AT2000_0250_0016.CC_Inputs.Current_actual_value_Ch[11] <-> CC Inputs/Current actual value Ch.12
//     PlcTask Inputs/GVL_iXlinker.EtherCAT_Master_ATxxxx.Beckhoff_AT1xxx.Beckhoff_AT2xxxEK1122.A_0004_AT2000_0250_0016.CC_Inputs.Current_actual_value_Ch[12] <-> CC Inputs/Current actual value Ch.13
//     PlcTask Inputs/GVL_iXlinker.EtherCAT_Master_ATxxxx.Beckhoff_AT1xxx.Beckhoff_AT2xxxEK1122.A_0004_AT2000_0250_0016.CC_Inputs.Current_actual_value_Ch[13] <-> CC Inputs/Current actual value Ch.14
//     PlcTask Inputs/GVL_iXlinker.EtherCAT_Master_ATxxxx.Beckhoff_AT1xxx.Beckhoff_AT2xxxEK1122.A_0004_AT2000_0250_0016.CC_Inputs.Current_actual_value_Ch[14] <-> CC Inputs/Current actual value Ch.15
//     PlcTask Outputs/GVL_iXlinker.EtherCAT_Master_ATxxxx.Beckhoff_AT1xxx.Beckhoff_AT2xxxEK1122.A_0004_AT2000_0250_0016.CC_Outputs.Control <-> CC Outputs/Control
//     PlcTask Outputs/GVL_iXlinker.EtherCAT_Master_ATxxxx.Beckhoff_AT1xxx.Beckhoff_AT2xxxEK1122.A_0004_AT2000_0250_0016.CC_Outputs.Current_setpoint_value_Ch[0] <-> CC Outputs/Current setpoint value Ch.1
//     PlcTask Outputs/GVL_iXlinker.EtherCAT_Master_ATxxxx.Beckhoff_AT1xxx.Beckhoff_AT2xxxEK1122.A_0004_AT2000_0250_0016.CC_Outputs.Current_setpoint_value_Ch[1] <-> CC Outputs/Current setpoint value Ch.2
//     PlcTask Outputs/GVL_iXlinker.EtherCAT_Master_ATxxxx.Beckhoff_AT1xxx.Beckhoff_AT2xxxEK1122.A_0004_AT2000_0250_0016.CC_Outputs.Current_setpoint_value_Ch[2] <-> CC Outputs/Current setpoint value Ch.3
//     PlcTask Outputs/GVL_iXlinker.EtherCAT_Master_ATxxxx.Beckhoff_AT1xxx.Beckhoff_AT2xxxEK1122.A_0004_AT2000_0250_0016.CC_Outputs.Current_setpoint_value_Ch[3] <-> CC Outputs/Current setpoint value Ch.4
//     PlcTask Outputs/GVL_iXlinker.EtherCAT_Master_ATxxxx.Beckhoff_AT1xxx.Beckhoff_AT2xxxEK1122.A_0004_AT2000_0250_0016.CC_Outputs.Current_setpoint_value_Ch[4] <-> CC Outputs/Current setpoint value Ch.5
//     PlcTask Outputs/GVL_iXlinker.EtherCAT_Master_ATxxxx.Beckhoff_AT1xxx.Beckhoff_AT2xxxEK1122.A_0004_AT2000_0250_0016.CC_Outputs.Current_setpoint_value_Ch[5] <-> CC Outputs/Current setpoint value Ch.6
//     PlcTask Outputs/GVL_iXlinker.EtherCAT_Master_ATxxxx.Beckhoff_AT1xxx.Beckhoff_AT2xxxEK1122.A_0004_AT2000_0250_0016.CC_Outputs.Current_setpoint_value_Ch[6] <-> CC Outputs/Current setpoint value Ch.7
//     PlcTask Outputs/GVL_iXlinker.EtherCAT_Master_ATxxxx.Beckhoff_AT1xxx.Beckhoff_AT2xxxEK1122.A_0004_AT2000_0250_0016.CC_Outputs.Current_setpoint_value_Ch[7] <-> CC Outputs/Current setpoint value Ch.8
//     PlcTask Outputs/GVL_iXlinker.EtherCAT_Master_ATxxxx.Beckhoff_AT1xxx.Beckhoff_AT2xxxEK1122.A_0004_AT2000_0250_0016.CC_Outputs.Current_setpoint_value_Ch[8] <-> CC Outputs/Current setpoint value Ch.9
//     PlcTask Outputs/GVL_iXlinker.EtherCAT_Master_ATxxxx.Beckhoff_AT1xxx.Beckhoff_AT2xxxEK1122.A_0004_AT2000_0250_0016.CC_Outputs.Current_setpoint_value_Ch[9] <-> CC Outputs/Current setpoint value Ch.10
//     PlcTask Outputs/GVL_iXlinker.EtherCAT_Master_ATxxxx.Beckhoff_AT1xxx.Beckhoff_AT2xxxEK1122.A_0004_AT2000_0250_0016.CC_Outputs.Current_setpoint_value_Ch[10] <-> CC Outputs/Current setpoint value Ch.11
//     PlcTask Outputs/GVL_iXlinker.EtherCAT_Master_ATxxxx.Beckhoff_AT1xxx.Beckhoff_AT2xxxEK1122.A_0004_AT2000_0250_0016.CC_Outputs.Current_setpoint_value_Ch[11] <-> CC Outputs/Current setpoint value Ch.12
//     PlcTask Outputs/GVL_iXlinker.EtherCAT_Master_ATxxxx.Beckhoff_AT1xxx.Beckhoff_AT2xxxEK1122.A_0004_AT2000_0250_0016.CC_Outputs.Current_setpoint_value_Ch[12] <-> CC Outputs/Current setpoint value Ch.13
//     PlcTask Outputs/GVL_iXlinker.EtherCAT_Master_ATxxxx.Beckhoff_AT1xxx.Beckhoff_AT2xxxEK1122.A_0004_AT2000_0250_0016.CC_Outputs.Current_setpoint_value_Ch[13] <-> CC Outputs/Current setpoint value Ch.14
//     PlcTask Outputs/GVL_iXlinker.EtherCAT_Master_ATxxxx.Beckhoff_AT1xxx.Beckhoff_AT2xxxEK1122.A_0004_AT2000_0250_0016.CC_Outputs.Current_setpoint_value_Ch[14] <-> CC Outputs/Current setpoint value Ch.15
//     PlcTask Inputs/GVL_iXlinker.EtherCAT_Master_ATxxxx.Beckhoff_AT1xxx.Beckhoff_AT2xxxEK1122.A_0004_AT2000_0250_0016.WcState.WcState <-> WcState/WcState
//     PlcTask Inputs/GVL_iXlinker.EtherCAT_Master_ATxxxx.Beckhoff_AT1xxx.Beckhoff_AT2xxxEK1122.A_0004_AT2000_0250_0016.WcState.InputToggle <-> WcState/InputToggle
//     PlcTask Inputs/GVL_iXlinker.EtherCAT_Master_ATxxxx.Beckhoff_AT1xxx.Beckhoff_AT2xxxEK1122.A_0004_AT2000_0250_0016.InfoData.AdsAddr <-> InfoData/AdsAddr
//     PlcTask Inputs/GVL_iXlinker.EtherCAT_Master_ATxxxx.Beckhoff_AT1xxx.Beckhoff_AT2xxxEK1122.A_0004_AT2000_0250_0016.InfoData.DcOutputShift <-> InfoData/DcOutputShift
//     PlcTask Inputs/GVL_iXlinker.EtherCAT_Master_ATxxxx.Beckhoff_AT1xxx.Beckhoff_AT2xxxEK1122.A_0004_AT2000_0250_0016.InfoData.DcInputShift <-> InfoData/DcInputShift
//     PlcTask Inputs/GVL_iXlinker.EtherCAT_Master_ATxxxx.Beckhoff_AT1xxx.Beckhoff_AT2xxxEK1122.A_0004_AT2000_0250_0016.InfoData.State <-> InfoData/State
//   PLC/PLC Instance <-> EtherCAT Master ATxxxx/Beckhoff AT1xxx/Beckhoff AT2xxxEK1122/A_0005(AT2000-0250-0017)
//     PlcTask Inputs/GVL_iXlinker.EtherCAT_Master_ATxxxx.Beckhoff_AT1xxx.Beckhoff_AT2xxxEK1122.A_0005_AT2000_0250_0017.CC_Inputs.Status <-> CC Inputs/Status
//     PlcTask Inputs/GVL_iXlinker.EtherCAT_Master_ATxxxx.Beckhoff_AT1xxx.Beckhoff_AT2xxxEK1122.A_0005_AT2000_0250_0017.CC_Inputs.Current_actual_value_Ch[0] <-> CC Inputs/Current actual value Ch.1
//     PlcTask Inputs/GVL_iXlinker.EtherCAT_Master_ATxxxx.Beckhoff_AT1xxx.Beckhoff_AT2xxxEK1122.A_0005_AT2000_0250_0017.CC_Inputs.Current_actual_value_Ch[1] <-> CC Inputs/Current actual value Ch.2
//     PlcTask Inputs/GVL_iXlinker.EtherCAT_Master_ATxxxx.Beckhoff_AT1xxx.Beckhoff_AT2xxxEK1122.A_0005_AT2000_0250_0017.CC_Inputs.Current_actual_value_Ch[2] <-> CC Inputs/Current actual value Ch.3
//     PlcTask Inputs/GVL_iXlinker.EtherCAT_Master_ATxxxx.Beckhoff_AT1xxx.Beckhoff_AT2xxxEK1122.A_0005_AT2000_0250_0017.CC_Inputs.Current_actual_value_Ch[3] <-> CC Inputs/Current actual value Ch.4
//     PlcTask Inputs/GVL_iXlinker.EtherCAT_Master_ATxxxx.Beckhoff_AT1xxx.Beckhoff_AT2xxxEK1122.A_0005_AT2000_0250_0017.CC_Inputs.Current_actual_value_Ch[4] <-> CC Inputs/Current actual value Ch.5
//     PlcTask Inputs/GVL_iXlinker.EtherCAT_Master_ATxxxx.Beckhoff_AT1xxx.Beckhoff_AT2xxxEK1122.A_0005_AT2000_0250_0017.CC_Inputs.Current_actual_value_Ch[5] <-> CC Inputs/Current actual value Ch.6
//     PlcTask Inputs/GVL_iXlinker.EtherCAT_Master_ATxxxx.Beckhoff_AT1xxx.Beckhoff_AT2xxxEK1122.A_0005_AT2000_0250_0017.CC_Inputs.Current_actual_value_Ch[6] <-> CC Inputs/Current actual value Ch.7
//     PlcTask Inputs/GVL_iXlinker.EtherCAT_Master_ATxxxx.Beckhoff_AT1xxx.Beckhoff_AT2xxxEK1122.A_0005_AT2000_0250_0017.CC_Inputs.Current_actual_value_Ch[7] <-> CC Inputs/Current actual value Ch.8
//     PlcTask Inputs/GVL_iXlinker.EtherCAT_Master_ATxxxx.Beckhoff_AT1xxx.Beckhoff_AT2xxxEK1122.A_0005_AT2000_0250_0017.CC_Inputs.Current_actual_value_Ch[8] <-> CC Inputs/Current actual value Ch.9
//     PlcTask Inputs/GVL_iXlinker.EtherCAT_Master_ATxxxx.Beckhoff_AT1xxx.Beckhoff_AT2xxxEK1122.A_0005_AT2000_0250_0017.CC_Inputs.Current_actual_value_Ch[9] <-> CC Inputs/Current actual value Ch.10
//     PlcTask Inputs/GVL_iXlinker.EtherCAT_Master_ATxxxx.Beckhoff_AT1xxx.Beckhoff_AT2xxxEK1122.A_0005_AT2000_0250_0017.CC_Inputs.Current_actual_value_Ch[10] <-> CC Inputs/Current actual value Ch.11
//     PlcTask Inputs/GVL_iXlinker.EtherCAT_Master_ATxxxx.Beckhoff_AT1xxx.Beckhoff_AT2xxxEK1122.A_0005_AT2000_0250_0017.CC_Inputs.Current_actual_value_Ch[11] <-> CC Inputs/Current actual value Ch.12
//     PlcTask Inputs/GVL_iXlinker.EtherCAT_Master_ATxxxx.Beckhoff_AT1xxx.Beckhoff_AT2xxxEK1122.A_0005_AT2000_0250_0017.CC_Inputs.Current_actual_value_Ch[12] <-> CC Inputs/Current actual value Ch.13
//     PlcTask Inputs/GVL_iXlinker.EtherCAT_Master_ATxxxx.Beckhoff_AT1xxx.Beckhoff_AT2xxxEK1122.A_0005_AT2000_0250_0017.CC_Inputs.Current_actual_value_Ch[13] <-> CC Inputs/Current actual value Ch.14
//     PlcTask Inputs/GVL_iXlinker.EtherCAT_Master_ATxxxx.Beckhoff_AT1xxx.Beckhoff_AT2xxxEK1122.A_0005_AT2000_0250_0017.CC_Inputs.Current_actual_value_Ch[14] <-> CC Inputs/Current actual value Ch.15
//     PlcTask Outputs/GVL_iXlinker.EtherCAT_Master_ATxxxx.Beckhoff_AT1xxx.Beckhoff_AT2xxxEK1122.A_0005_AT2000_0250_0017.CC_Outputs.Control <-> CC Outputs/Control
//     PlcTask Outputs/GVL_iXlinker.EtherCAT_Master_ATxxxx.Beckhoff_AT1xxx.Beckhoff_AT2xxxEK1122.A_0005_AT2000_0250_0017.CC_Outputs.Current_setpoint_value_Ch[0] <-> CC Outputs/Current setpoint value Ch.1
//     PlcTask Outputs/GVL_iXlinker.EtherCAT_Master_ATxxxx.Beckhoff_AT1xxx.Beckhoff_AT2xxxEK1122.A_0005_AT2000_0250_0017.CC_Outputs.Current_setpoint_value_Ch[1] <-> CC Outputs/Current setpoint value Ch.2
//     PlcTask Outputs/GVL_iXlinker.EtherCAT_Master_ATxxxx.Beckhoff_AT1xxx.Beckhoff_AT2xxxEK1122.A_0005_AT2000_0250_0017.CC_Outputs.Current_setpoint_value_Ch[2] <-> CC Outputs/Current setpoint value Ch.3
//     PlcTask Outputs/GVL_iXlinker.EtherCAT_Master_ATxxxx.Beckhoff_AT1xxx.Beckhoff_AT2xxxEK1122.A_0005_AT2000_0250_0017.CC_Outputs.Current_setpoint_value_Ch[3] <-> CC Outputs/Current setpoint value Ch.4
//     PlcTask Outputs/GVL_iXlinker.EtherCAT_Master_ATxxxx.Beckhoff_AT1xxx.Beckhoff_AT2xxxEK1122.A_0005_AT2000_0250_0017.CC_Outputs.Current_setpoint_value_Ch[4] <-> CC Outputs/Current setpoint value Ch.5
//     PlcTask Outputs/GVL_iXlinker.EtherCAT_Master_ATxxxx.Beckhoff_AT1xxx.Beckhoff_AT2xxxEK1122.A_0005_AT2000_0250_0017.CC_Outputs.Current_setpoint_value_Ch[5] <-> CC Outputs/Current setpoint value Ch.6
//     PlcTask Outputs/GVL_iXlinker.EtherCAT_Master_ATxxxx.Beckhoff_AT1xxx.Beckhoff_AT2xxxEK1122.A_0005_AT2000_0250_0017.CC_Outputs.Current_setpoint_value_Ch[6] <-> CC Outputs/Current setpoint value Ch.7
//     PlcTask Outputs/GVL_iXlinker.EtherCAT_Master_ATxxxx.Beckhoff_AT1xxx.Beckhoff_AT2xxxEK1122.A_0005_AT2000_0250_0017.CC_Outputs.Current_setpoint_value_Ch[7] <-> CC Outputs/Current setpoint value Ch.8
//     PlcTask Outputs/GVL_iXlinker.EtherCAT_Master_ATxxxx.Beckhoff_AT1xxx.Beckhoff_AT2xxxEK1122.A_0005_AT2000_0250_0017.CC_Outputs.Current_setpoint_value_Ch[8] <-> CC Outputs/Current setpoint value Ch.9
//     PlcTask Outputs/GVL_iXlinker.EtherCAT_Master_ATxxxx.Beckhoff_AT1xxx.Beckhoff_AT2xxxEK1122.A_0005_AT2000_0250_0017.CC_Outputs.Current_setpoint_value_Ch[9] <-> CC Outputs/Current setpoint value Ch.10
//     PlcTask Outputs/GVL_iXlinker.EtherCAT_Master_ATxxxx.Beckhoff_AT1xxx.Beckhoff_AT2xxxEK1122.A_0005_AT2000_0250_0017.CC_Outputs.Current_setpoint_value_Ch[10] <-> CC Outputs/Current setpoint value Ch.11
//     PlcTask Outputs/GVL_iXlinker.EtherCAT_Master_ATxxxx.Beckhoff_AT1xxx.Beckhoff_AT2xxxEK1122.A_0005_AT2000_0250_0017.CC_Outputs.Current_setpoint_value_Ch[11] <-> CC Outputs/Current setpoint value Ch.12
//     PlcTask Outputs/GVL_iXlinker.EtherCAT_Master_ATxxxx.Beckhoff_AT1xxx.Beckhoff_AT2xxxEK1122.A_0005_AT2000_0250_0017.CC_Outputs.Current_setpoint_value_Ch[12] <-> CC Outputs/Current setpoint value Ch.13
//     PlcTask Outputs/GVL_iXlinker.EtherCAT_Master_ATxxxx.Beckhoff_AT1xxx.Beckhoff_AT2xxxEK1122.A_0005_AT2000_0250_0017.CC_Outputs.Current_setpoint_value_Ch[13] <-> CC Outputs/Current setpoint value Ch.14
//     PlcTask Outputs/GVL_iXlinker.EtherCAT_Master_ATxxxx.Beckhoff_AT1xxx.Beckhoff_AT2xxxEK1122.A_0005_AT2000_0250_0017.CC_Outputs.Current_setpoint_value_Ch[14] <-> CC Outputs/Current setpoint value Ch.15
//     PlcTask Inputs/GVL_iXlinker.EtherCAT_Master_ATxxxx.Beckhoff_AT1xxx.Beckhoff_AT2xxxEK1122.A_0005_AT2000_0250_0017.WcState.WcState <-> WcState/WcState
//     PlcTask Inputs/GVL_iXlinker.EtherCAT_Master_ATxxxx.Beckhoff_AT1xxx.Beckhoff_AT2xxxEK1122.A_0005_AT2000_0250_0017.WcState.InputToggle <-> WcState/InputToggle
//     PlcTask Inputs/GVL_iXlinker.EtherCAT_Master_ATxxxx.Beckhoff_AT1xxx.Beckhoff_AT2xxxEK1122.A_0005_AT2000_0250_0017.InfoData.AdsAddr <-> InfoData/AdsAddr
//     PlcTask Inputs/GVL_iXlinker.EtherCAT_Master_ATxxxx.Beckhoff_AT1xxx.Beckhoff_AT2xxxEK1122.A_0005_AT2000_0250_0017.InfoData.DcOutputShift <-> InfoData/DcOutputShift
//     PlcTask Inputs/GVL_iXlinker.EtherCAT_Master_ATxxxx.Beckhoff_AT1xxx.Beckhoff_AT2xxxEK1122.A_0005_AT2000_0250_0017.InfoData.DcInputShift <-> InfoData/DcInputShift
//     PlcTask Inputs/GVL_iXlinker.EtherCAT_Master_ATxxxx.Beckhoff_AT1xxx.Beckhoff_AT2xxxEK1122.A_0005_AT2000_0250_0017.InfoData.State <-> InfoData/State
//   PLC/PLC Instance <-> EtherCAT Master ATxxxx/Beckhoff AT1xxx/Beckhoff AT2xxxEK1122/A_0006(AT2000-0250-0018)
//     PlcTask Inputs/GVL_iXlinker.EtherCAT_Master_ATxxxx.Beckhoff_AT1xxx.Beckhoff_AT2xxxEK1122.A_0006_AT2000_0250_0018.CC_Inputs.Status <-> CC Inputs/Status
//     PlcTask Inputs/GVL_iXlinker.EtherCAT_Master_ATxxxx.Beckhoff_AT1xxx.Beckhoff_AT2xxxEK1122.A_0006_AT2000_0250_0018.CC_Inputs.Current_actual_value_Ch[0] <-> CC Inputs/Current actual value Ch.1
//     PlcTask Inputs/GVL_iXlinker.EtherCAT_Master_ATxxxx.Beckhoff_AT1xxx.Beckhoff_AT2xxxEK1122.A_0006_AT2000_0250_0018.CC_Inputs.Current_actual_value_Ch[1] <-> CC Inputs/Current actual value Ch.2
//     PlcTask Inputs/GVL_iXlinker.EtherCAT_Master_ATxxxx.Beckhoff_AT1xxx.Beckhoff_AT2xxxEK1122.A_0006_AT2000_0250_0018.CC_Inputs.Current_actual_value_Ch[2] <-> CC Inputs/Current actual value Ch.3
//     PlcTask Inputs/GVL_iXlinker.EtherCAT_Master_ATxxxx.Beckhoff_AT1xxx.Beckhoff_AT2xxxEK1122.A_0006_AT2000_0250_0018.CC_Inputs.Current_actual_value_Ch[3] <-> CC Inputs/Current actual value Ch.4
//     PlcTask Inputs/GVL_iXlinker.EtherCAT_Master_ATxxxx.Beckhoff_AT1xxx.Beckhoff_AT2xxxEK1122.A_0006_AT2000_0250_0018.CC_Inputs.Current_actual_value_Ch[4] <-> CC Inputs/Current actual value Ch.5
//     PlcTask Inputs/GVL_iXlinker.EtherCAT_Master_ATxxxx.Beckhoff_AT1xxx.Beckhoff_AT2xxxEK1122.A_0006_AT2000_0250_0018.CC_Inputs.Current_actual_value_Ch[5] <-> CC Inputs/Current actual value Ch.6
//     PlcTask Inputs/GVL_iXlinker.EtherCAT_Master_ATxxxx.Beckhoff_AT1xxx.Beckhoff_AT2xxxEK1122.A_0006_AT2000_0250_0018.CC_Inputs.Current_actual_value_Ch[6] <-> CC Inputs/Current actual value Ch.7
//     PlcTask Inputs/GVL_iXlinker.EtherCAT_Master_ATxxxx.Beckhoff_AT1xxx.Beckhoff_AT2xxxEK1122.A_0006_AT2000_0250_0018.CC_Inputs.Current_actual_value_Ch[7] <-> CC Inputs/Current actual value Ch.8
//     PlcTask Inputs/GVL_iXlinker.EtherCAT_Master_ATxxxx.Beckhoff_AT1xxx.Beckhoff_AT2xxxEK1122.A_0006_AT2000_0250_0018.CC_Inputs.Current_actual_value_Ch[8] <-> CC Inputs/Current actual value Ch.9
//     PlcTask Inputs/GVL_iXlinker.EtherCAT_Master_ATxxxx.Beckhoff_AT1xxx.Beckhoff_AT2xxxEK1122.A_0006_AT2000_0250_0018.CC_Inputs.Current_actual_value_Ch[9] <-> CC Inputs/Current actual value Ch.10
//     PlcTask Inputs/GVL_iXlinker.EtherCAT_Master_ATxxxx.Beckhoff_AT1xxx.Beckhoff_AT2xxxEK1122.A_0006_AT2000_0250_0018.CC_Inputs.Current_actual_value_Ch[10] <-> CC Inputs/Current actual value Ch.11
//     PlcTask Inputs/GVL_iXlinker.EtherCAT_Master_ATxxxx.Beckhoff_AT1xxx.Beckhoff_AT2xxxEK1122.A_0006_AT2000_0250_0018.CC_Inputs.Current_actual_value_Ch[11] <-> CC Inputs/Current actual value Ch.12
//     PlcTask Inputs/GVL_iXlinker.EtherCAT_Master_ATxxxx.Beckhoff_AT1xxx.Beckhoff_AT2xxxEK1122.A_0006_AT2000_0250_0018.CC_Inputs.Current_actual_value_Ch[12] <-> CC Inputs/Current actual value Ch.13
//     PlcTask Inputs/GVL_iXlinker.EtherCAT_Master_ATxxxx.Beckhoff_AT1xxx.Beckhoff_AT2xxxEK1122.A_0006_AT2000_0250_0018.CC_Inputs.Current_actual_value_Ch[13] <-> CC Inputs/Current actual value Ch.14
//     PlcTask Inputs/GVL_iXlinker.EtherCAT_Master_ATxxxx.Beckhoff_AT1xxx.Beckhoff_AT2xxxEK1122.A_0006_AT2000_0250_0018.CC_Inputs.Current_actual_value_Ch[14] <-> CC Inputs/Current actual value Ch.15
//     PlcTask Outputs/GVL_iXlinker.EtherCAT_Master_ATxxxx.Beckhoff_AT1xxx.Beckhoff_AT2xxxEK1122.A_0006_AT2000_0250_0018.CC_Outputs.Control <-> CC Outputs/Control
//     PlcTask Outputs/GVL_iXlinker.EtherCAT_Master_ATxxxx.Beckhoff_AT1xxx.Beckhoff_AT2xxxEK1122.A_0006_AT2000_0250_0018.CC_Outputs.Current_setpoint_value_Ch[0] <-> CC Outputs/Current setpoint value Ch.1
//     PlcTask Outputs/GVL_iXlinker.EtherCAT_Master_ATxxxx.Beckhoff_AT1xxx.Beckhoff_AT2xxxEK1122.A_0006_AT2000_0250_0018.CC_Outputs.Current_setpoint_value_Ch[1] <-> CC Outputs/Current setpoint value Ch.2
//     PlcTask Outputs/GVL_iXlinker.EtherCAT_Master_ATxxxx.Beckhoff_AT1xxx.Beckhoff_AT2xxxEK1122.A_0006_AT2000_0250_0018.CC_Outputs.Current_setpoint_value_Ch[2] <-> CC Outputs/Current setpoint value Ch.3
//     PlcTask Outputs/GVL_iXlinker.EtherCAT_Master_ATxxxx.Beckhoff_AT1xxx.Beckhoff_AT2xxxEK1122.A_0006_AT2000_0250_0018.CC_Outputs.Current_setpoint_value_Ch[3] <-> CC Outputs/Current setpoint value Ch.4
//     PlcTask Outputs/GVL_iXlinker.EtherCAT_Master_ATxxxx.Beckhoff_AT1xxx.Beckhoff_AT2xxxEK1122.A_0006_AT2000_0250_0018.CC_Outputs.Current_setpoint_value_Ch[4] <-> CC Outputs/Current setpoint value Ch.5
//     PlcTask Outputs/GVL_iXlinker.EtherCAT_Master_ATxxxx.Beckhoff_AT1xxx.Beckhoff_AT2xxxEK1122.A_0006_AT2000_0250_0018.CC_Outputs.Current_setpoint_value_Ch[5] <-> CC Outputs/Current setpoint value Ch.6
//     PlcTask Outputs/GVL_iXlinker.EtherCAT_Master_ATxxxx.Beckhoff_AT1xxx.Beckhoff_AT2xxxEK1122.A_0006_AT2000_0250_0018.CC_Outputs.Current_setpoint_value_Ch[6] <-> CC Outputs/Current setpoint value Ch.7
//     PlcTask Outputs/GVL_iXlinker.EtherCAT_Master_ATxxxx.Beckhoff_AT1xxx.Beckhoff_AT2xxxEK1122.A_0006_AT2000_0250_0018.CC_Outputs.Current_setpoint_value_Ch[7] <-> CC Outputs/Current setpoint value Ch.8
//     PlcTask Outputs/GVL_iXlinker.EtherCAT_Master_ATxxxx.Beckhoff_AT1xxx.Beckhoff_AT2xxxEK1122.A_0006_AT2000_0250_0018.CC_Outputs.Current_setpoint_value_Ch[8] <-> CC Outputs/Current setpoint value Ch.9
//     PlcTask Outputs/GVL_iXlinker.EtherCAT_Master_ATxxxx.Beckhoff_AT1xxx.Beckhoff_AT2xxxEK1122.A_0006_AT2000_0250_0018.CC_Outputs.Current_setpoint_value_Ch[9] <-> CC Outputs/Current setpoint value Ch.10
//     PlcTask Outputs/GVL_iXlinker.EtherCAT_Master_ATxxxx.Beckhoff_AT1xxx.Beckhoff_AT2xxxEK1122.A_0006_AT2000_0250_0018.CC_Outputs.Current_setpoint_value_Ch[10] <-> CC Outputs/Current setpoint value Ch.11
//     PlcTask Outputs/GVL_iXlinker.EtherCAT_Master_ATxxxx.Beckhoff_AT1xxx.Beckhoff_AT2xxxEK1122.A_0006_AT2000_0250_0018.CC_Outputs.Current_setpoint_value_Ch[11] <-> CC Outputs/Current setpoint value Ch.12
//     PlcTask Outputs/GVL_iXlinker.EtherCAT_Master_ATxxxx.Beckhoff_AT1xxx.Beckhoff_AT2xxxEK1122.A_0006_AT2000_0250_0018.CC_Outputs.Current_setpoint_value_Ch[12] <-> CC Outputs/Current setpoint value Ch.13
//     PlcTask Outputs/GVL_iXlinker.EtherCAT_Master_ATxxxx.Beckhoff_AT1xxx.Beckhoff_AT2xxxEK1122.A_0006_AT2000_0250_0018.CC_Outputs.Current_setpoint_value_Ch[13] <-> CC Outputs/Current setpoint value Ch.14
//     PlcTask Outputs/GVL_iXlinker.EtherCAT_Master_ATxxxx.Beckhoff_AT1xxx.Beckhoff_AT2xxxEK1122.A_0006_AT2000_0250_0018.CC_Outputs.Current_setpoint_value_Ch[14] <-> CC Outputs/Current setpoint value Ch.15
//     PlcTask Inputs/GVL_iXlinker.EtherCAT_Master_ATxxxx.Beckhoff_AT1xxx.Beckhoff_AT2xxxEK1122.A_0006_AT2000_0250_0018.WcState.WcState <-> WcState/WcState
//     PlcTask Inputs/GVL_iXlinker.EtherCAT_Master_ATxxxx.Beckhoff_AT1xxx.Beckhoff_AT2xxxEK1122.A_0006_AT2000_0250_0018.WcState.InputToggle <-> WcState/InputToggle
//     PlcTask Inputs/GVL_iXlinker.EtherCAT_Master_ATxxxx.Beckhoff_AT1xxx.Beckhoff_AT2xxxEK1122.A_0006_AT2000_0250_0018.InfoData.AdsAddr <-> InfoData/AdsAddr
//     PlcTask Inputs/GVL_iXlinker.EtherCAT_Master_ATxxxx.Beckhoff_AT1xxx.Beckhoff_AT2xxxEK1122.A_0006_AT2000_0250_0018.InfoData.DcOutputShift <-> InfoData/DcOutputShift
//     PlcTask Inputs/GVL_iXlinker.EtherCAT_Master_ATxxxx.Beckhoff_AT1xxx.Beckhoff_AT2xxxEK1122.A_0006_AT2000_0250_0018.InfoData.DcInputShift <-> InfoData/DcInputShift
//     PlcTask Inputs/GVL_iXlinker.EtherCAT_Master_ATxxxx.Beckhoff_AT1xxx.Beckhoff_AT2xxxEK1122.A_0006_AT2000_0250_0018.InfoData.State <-> InfoData/State
//   PLC/PLC Instance <-> EtherCAT Master ATxxxx/Beckhoff AT1xxx/Beckhoff AT2xxxEK1122/A_0007(AT2000-0250-0019)
//     PlcTask Inputs/GVL_iXlinker.EtherCAT_Master_ATxxxx.Beckhoff_AT1xxx.Beckhoff_AT2xxxEK1122.A_0007_AT2000_0250_0019.CC_Inputs.Status <-> CC Inputs/Status
//     PlcTask Inputs/GVL_iXlinker.EtherCAT_Master_ATxxxx.Beckhoff_AT1xxx.Beckhoff_AT2xxxEK1122.A_0007_AT2000_0250_0019.CC_Inputs.Current_actual_value_Ch[0] <-> CC Inputs/Current actual value Ch.1
//     PlcTask Inputs/GVL_iXlinker.EtherCAT_Master_ATxxxx.Beckhoff_AT1xxx.Beckhoff_AT2xxxEK1122.A_0007_AT2000_0250_0019.CC_Inputs.Current_actual_value_Ch[1] <-> CC Inputs/Current actual value Ch.2
//     PlcTask Inputs/GVL_iXlinker.EtherCAT_Master_ATxxxx.Beckhoff_AT1xxx.Beckhoff_AT2xxxEK1122.A_0007_AT2000_0250_0019.CC_Inputs.Current_actual_value_Ch[2] <-> CC Inputs/Current actual value Ch.3
//     PlcTask Inputs/GVL_iXlinker.EtherCAT_Master_ATxxxx.Beckhoff_AT1xxx.Beckhoff_AT2xxxEK1122.A_0007_AT2000_0250_0019.CC_Inputs.Current_actual_value_Ch[3] <-> CC Inputs/Current actual value Ch.4
//     PlcTask Inputs/GVL_iXlinker.EtherCAT_Master_ATxxxx.Beckhoff_AT1xxx.Beckhoff_AT2xxxEK1122.A_0007_AT2000_0250_0019.CC_Inputs.Current_actual_value_Ch[4] <-> CC Inputs/Current actual value Ch.5
//     PlcTask Inputs/GVL_iXlinker.EtherCAT_Master_ATxxxx.Beckhoff_AT1xxx.Beckhoff_AT2xxxEK1122.A_0007_AT2000_0250_0019.CC_Inputs.Current_actual_value_Ch[5] <-> CC Inputs/Current actual value Ch.6
//     PlcTask Inputs/GVL_iXlinker.EtherCAT_Master_ATxxxx.Beckhoff_AT1xxx.Beckhoff_AT2xxxEK1122.A_0007_AT2000_0250_0019.CC_Inputs.Current_actual_value_Ch[6] <-> CC Inputs/Current actual value Ch.7
//     PlcTask Inputs/GVL_iXlinker.EtherCAT_Master_ATxxxx.Beckhoff_AT1xxx.Beckhoff_AT2xxxEK1122.A_0007_AT2000_0250_0019.CC_Inputs.Current_actual_value_Ch[7] <-> CC Inputs/Current actual value Ch.8
//     PlcTask Inputs/GVL_iXlinker.EtherCAT_Master_ATxxxx.Beckhoff_AT1xxx.Beckhoff_AT2xxxEK1122.A_0007_AT2000_0250_0019.CC_Inputs.Current_actual_value_Ch[8] <-> CC Inputs/Current actual value Ch.9
//     PlcTask Inputs/GVL_iXlinker.EtherCAT_Master_ATxxxx.Beckhoff_AT1xxx.Beckhoff_AT2xxxEK1122.A_0007_AT2000_0250_0019.CC_Inputs.Current_actual_value_Ch[9] <-> CC Inputs/Current actual value Ch.10
//     PlcTask Inputs/GVL_iXlinker.EtherCAT_Master_ATxxxx.Beckhoff_AT1xxx.Beckhoff_AT2xxxEK1122.A_0007_AT2000_0250_0019.CC_Inputs.Current_actual_value_Ch[10] <-> CC Inputs/Current actual value Ch.11
//     PlcTask Inputs/GVL_iXlinker.EtherCAT_Master_ATxxxx.Beckhoff_AT1xxx.Beckhoff_AT2xxxEK1122.A_0007_AT2000_0250_0019.CC_Inputs.Current_actual_value_Ch[11] <-> CC Inputs/Current actual value Ch.12
//     PlcTask Inputs/GVL_iXlinker.EtherCAT_Master_ATxxxx.Beckhoff_AT1xxx.Beckhoff_AT2xxxEK1122.A_0007_AT2000_0250_0019.CC_Inputs.Current_actual_value_Ch[12] <-> CC Inputs/Current actual value Ch.13
//     PlcTask Inputs/GVL_iXlinker.EtherCAT_Master_ATxxxx.Beckhoff_AT1xxx.Beckhoff_AT2xxxEK1122.A_0007_AT2000_0250_0019.CC_Inputs.Current_actual_value_Ch[13] <-> CC Inputs/Current actual value Ch.14
//     PlcTask Inputs/GVL_iXlinker.EtherCAT_Master_ATxxxx.Beckhoff_AT1xxx.Beckhoff_AT2xxxEK1122.A_0007_AT2000_0250_0019.CC_Inputs.Current_actual_value_Ch[14] <-> CC Inputs/Current actual value Ch.15
//     PlcTask Outputs/GVL_iXlinker.EtherCAT_Master_ATxxxx.Beckhoff_AT1xxx.Beckhoff_AT2xxxEK1122.A_0007_AT2000_0250_0019.CC_Outputs.Control <-> CC Outputs/Control
//     PlcTask Outputs/GVL_iXlinker.EtherCAT_Master_ATxxxx.Beckhoff_AT1xxx.Beckhoff_AT2xxxEK1122.A_0007_AT2000_0250_0019.CC_Outputs.Current_setpoint_value_Ch[0] <-> CC Outputs/Current setpoint value Ch.1
//     PlcTask Outputs/GVL_iXlinker.EtherCAT_Master_ATxxxx.Beckhoff_AT1xxx.Beckhoff_AT2xxxEK1122.A_0007_AT2000_0250_0019.CC_Outputs.Current_setpoint_value_Ch[1] <-> CC Outputs/Current setpoint value Ch.2
//     PlcTask Outputs/GVL_iXlinker.EtherCAT_Master_ATxxxx.Beckhoff_AT1xxx.Beckhoff_AT2xxxEK1122.A_0007_AT2000_0250_0019.CC_Outputs.Current_setpoint_value_Ch[2] <-> CC Outputs/Current setpoint value Ch.3
//     PlcTask Outputs/GVL_iXlinker.EtherCAT_Master_ATxxxx.Beckhoff_AT1xxx.Beckhoff_AT2xxxEK1122.A_0007_AT2000_0250_0019.CC_Outputs.Current_setpoint_value_Ch[3] <-> CC Outputs/Current setpoint value Ch.4
//     PlcTask Outputs/GVL_iXlinker.EtherCAT_Master_ATxxxx.Beckhoff_AT1xxx.Beckhoff_AT2xxxEK1122.A_0007_AT2000_0250_0019.CC_Outputs.Current_setpoint_value_Ch[4] <-> CC Outputs/Current setpoint value Ch.5
//     PlcTask Outputs/GVL_iXlinker.EtherCAT_Master_ATxxxx.Beckhoff_AT1xxx.Beckhoff_AT2xxxEK1122.A_0007_AT2000_0250_0019.CC_Outputs.Current_setpoint_value_Ch[5] <-> CC Outputs/Current setpoint value Ch.6
//     PlcTask Outputs/GVL_iXlinker.EtherCAT_Master_ATxxxx.Beckhoff_AT1xxx.Beckhoff_AT2xxxEK1122.A_0007_AT2000_0250_0019.CC_Outputs.Current_setpoint_value_Ch[6] <-> CC Outputs/Current setpoint value Ch.7
//     PlcTask Outputs/GVL_iXlinker.EtherCAT_Master_ATxxxx.Beckhoff_AT1xxx.Beckhoff_AT2xxxEK1122.A_0007_AT2000_0250_0019.CC_Outputs.Current_setpoint_value_Ch[7] <-> CC Outputs/Current setpoint value Ch.8
//     PlcTask Outputs/GVL_iXlinker.EtherCAT_Master_ATxxxx.Beckhoff_AT1xxx.Beckhoff_AT2xxxEK1122.A_0007_AT2000_0250_0019.CC_Outputs.Current_setpoint_value_Ch[8] <-> CC Outputs/Current setpoint value Ch.9
//     PlcTask Outputs/GVL_iXlinker.EtherCAT_Master_ATxxxx.Beckhoff_AT1xxx.Beckhoff_AT2xxxEK1122.A_0007_AT2000_0250_0019.CC_Outputs.Current_setpoint_value_Ch[9] <-> CC Outputs/Current setpoint value Ch.10
//     PlcTask Outputs/GVL_iXlinker.EtherCAT_Master_ATxxxx.Beckhoff_AT1xxx.Beckhoff_AT2xxxEK1122.A_0007_AT2000_0250_0019.CC_Outputs.Current_setpoint_value_Ch[10] <-> CC Outputs/Current setpoint value Ch.11
//     PlcTask Outputs/GVL_iXlinker.EtherCAT_Master_ATxxxx.Beckhoff_AT1xxx.Beckhoff_AT2xxxEK1122.A_0007_AT2000_0250_0019.CC_Outputs.Current_setpoint_value_Ch[11] <-> CC Outputs/Current setpoint value Ch.12
//     PlcTask Outputs/GVL_iXlinker.EtherCAT_Master_ATxxxx.Beckhoff_AT1xxx.Beckhoff_AT2xxxEK1122.A_0007_AT2000_0250_0019.CC_Outputs.Current_setpoint_value_Ch[12] <-> CC Outputs/Current setpoint value Ch.13
//     PlcTask Outputs/GVL_iXlinker.EtherCAT_Master_ATxxxx.Beckhoff_AT1xxx.Beckhoff_AT2xxxEK1122.A_0007_AT2000_0250_0019.CC_Outputs.Current_setpoint_value_Ch[13] <-> CC Outputs/Current setpoint value Ch.14
//     PlcTask Outputs/GVL_iXlinker.EtherCAT_Master_ATxxxx.Beckhoff_AT1xxx.Beckhoff_AT2xxxEK1122.A_0007_AT2000_0250_0019.CC_Outputs.Current_setpoint_value_Ch[14] <-> CC Outputs/Current setpoint value Ch.15
//     PlcTask Inputs/GVL_iXlinker.EtherCAT_Master_ATxxxx.Beckhoff_AT1xxx.Beckhoff_AT2xxxEK1122.A_0007_AT2000_0250_0019.WcState.WcState <-> WcState/WcState
//     PlcTask Inputs/GVL_iXlinker.EtherCAT_Master_ATxxxx.Beckhoff_AT1xxx.Beckhoff_AT2xxxEK1122.A_0007_AT2000_0250_0019.WcState.InputToggle <-> WcState/InputToggle
//     PlcTask Inputs/GVL_iXlinker.EtherCAT_Master_ATxxxx.Beckhoff_AT1xxx.Beckhoff_AT2xxxEK1122.A_0007_AT2000_0250_0019.InfoData.AdsAddr <-> InfoData/AdsAddr
//     PlcTask Inputs/GVL_iXlinker.EtherCAT_Master_ATxxxx.Beckhoff_AT1xxx.Beckhoff_AT2xxxEK1122.A_0007_AT2000_0250_0019.InfoData.DcOutputShift <-> InfoData/DcOutputShift
//     PlcTask Inputs/GVL_iXlinker.EtherCAT_Master_ATxxxx.Beckhoff_AT1xxx.Beckhoff_AT2xxxEK1122.A_0007_AT2000_0250_0019.InfoData.DcInputShift <-> InfoData/DcInputShift
//     PlcTask Inputs/GVL_iXlinker.EtherCAT_Master_ATxxxx.Beckhoff_AT1xxx.Beckhoff_AT2xxxEK1122.A_0007_AT2000_0250_0019.InfoData.State <-> InfoData/State
//   PLC/PLC Instance <-> EtherCAT Master ATxxxx/Beckhoff AT1xxx/Beckhoff AT2xxxEK1122/A_0008(AT2000-0250-0020)
//     PlcTask Inputs/GVL_iXlinker.EtherCAT_Master_ATxxxx.Beckhoff_AT1xxx.Beckhoff_AT2xxxEK1122.A_0008_AT2000_0250_0020.CC_Inputs.Status <-> CC Inputs/Status
//     PlcTask Inputs/GVL_iXlinker.EtherCAT_Master_ATxxxx.Beckhoff_AT1xxx.Beckhoff_AT2xxxEK1122.A_0008_AT2000_0250_0020.CC_Inputs.Current_actual_value_Ch[0] <-> CC Inputs/Current actual value Ch.1
//     PlcTask Inputs/GVL_iXlinker.EtherCAT_Master_ATxxxx.Beckhoff_AT1xxx.Beckhoff_AT2xxxEK1122.A_0008_AT2000_0250_0020.CC_Inputs.Current_actual_value_Ch[1] <-> CC Inputs/Current actual value Ch.2
//     PlcTask Inputs/GVL_iXlinker.EtherCAT_Master_ATxxxx.Beckhoff_AT1xxx.Beckhoff_AT2xxxEK1122.A_0008_AT2000_0250_0020.CC_Inputs.Current_actual_value_Ch[2] <-> CC Inputs/Current actual value Ch.3
//     PlcTask Inputs/GVL_iXlinker.EtherCAT_Master_ATxxxx.Beckhoff_AT1xxx.Beckhoff_AT2xxxEK1122.A_0008_AT2000_0250_0020.CC_Inputs.Current_actual_value_Ch[3] <-> CC Inputs/Current actual value Ch.4
//     PlcTask Inputs/GVL_iXlinker.EtherCAT_Master_ATxxxx.Beckhoff_AT1xxx.Beckhoff_AT2xxxEK1122.A_0008_AT2000_0250_0020.CC_Inputs.Current_actual_value_Ch[4] <-> CC Inputs/Current actual value Ch.5
//     PlcTask Inputs/GVL_iXlinker.EtherCAT_Master_ATxxxx.Beckhoff_AT1xxx.Beckhoff_AT2xxxEK1122.A_0008_AT2000_0250_0020.CC_Inputs.Current_actual_value_Ch[5] <-> CC Inputs/Current actual value Ch.6
//     PlcTask Inputs/GVL_iXlinker.EtherCAT_Master_ATxxxx.Beckhoff_AT1xxx.Beckhoff_AT2xxxEK1122.A_0008_AT2000_0250_0020.CC_Inputs.Current_actual_value_Ch[6] <-> CC Inputs/Current actual value Ch.7
//     PlcTask Inputs/GVL_iXlinker.EtherCAT_Master_ATxxxx.Beckhoff_AT1xxx.Beckhoff_AT2xxxEK1122.A_0008_AT2000_0250_0020.CC_Inputs.Current_actual_value_Ch[7] <-> CC Inputs/Current actual value Ch.8
//     PlcTask Inputs/GVL_iXlinker.EtherCAT_Master_ATxxxx.Beckhoff_AT1xxx.Beckhoff_AT2xxxEK1122.A_0008_AT2000_0250_0020.CC_Inputs.Current_actual_value_Ch[8] <-> CC Inputs/Current actual value Ch.9
//     PlcTask Inputs/GVL_iXlinker.EtherCAT_Master_ATxxxx.Beckhoff_AT1xxx.Beckhoff_AT2xxxEK1122.A_0008_AT2000_0250_0020.CC_Inputs.Current_actual_value_Ch[9] <-> CC Inputs/Current actual value Ch.10
//     PlcTask Inputs/GVL_iXlinker.EtherCAT_Master_ATxxxx.Beckhoff_AT1xxx.Beckhoff_AT2xxxEK1122.A_0008_AT2000_0250_0020.CC_Inputs.Current_actual_value_Ch[10] <-> CC Inputs/Current actual value Ch.11
//     PlcTask Inputs/GVL_iXlinker.EtherCAT_Master_ATxxxx.Beckhoff_AT1xxx.Beckhoff_AT2xxxEK1122.A_0008_AT2000_0250_0020.CC_Inputs.Current_actual_value_Ch[11] <-> CC Inputs/Current actual value Ch.12
//     PlcTask Inputs/GVL_iXlinker.EtherCAT_Master_ATxxxx.Beckhoff_AT1xxx.Beckhoff_AT2xxxEK1122.A_0008_AT2000_0250_0020.CC_Inputs.Current_actual_value_Ch[12] <-> CC Inputs/Current actual value Ch.13
//     PlcTask Inputs/GVL_iXlinker.EtherCAT_Master_ATxxxx.Beckhoff_AT1xxx.Beckhoff_AT2xxxEK1122.A_0008_AT2000_0250_0020.CC_Inputs.Current_actual_value_Ch[13] <-> CC Inputs/Current actual value Ch.14
//     PlcTask Inputs/GVL_iXlinker.EtherCAT_Master_ATxxxx.Beckhoff_AT1xxx.Beckhoff_AT2xxxEK1122.A_0008_AT2000_0250_0020.CC_Inputs.Current_actual_value_Ch[14] <-> CC Inputs/Current actual value Ch.15
//     PlcTask Outputs/GVL_iXlinker.EtherCAT_Master_ATxxxx.Beckhoff_AT1xxx.Beckhoff_AT2xxxEK1122.A_0008_AT2000_0250_0020.CC_Outputs.Control <-> CC Outputs/Control
//     PlcTask Outputs/GVL_iXlinker.EtherCAT_Master_ATxxxx.Beckhoff_AT1xxx.Beckhoff_AT2xxxEK1122.A_0008_AT2000_0250_0020.CC_Outputs.Current_setpoint_value_Ch[0] <-> CC Outputs/Current setpoint value Ch.1
//     PlcTask Outputs/GVL_iXlinker.EtherCAT_Master_ATxxxx.Beckhoff_AT1xxx.Beckhoff_AT2xxxEK1122.A_0008_AT2000_0250_0020.CC_Outputs.Current_setpoint_value_Ch[1] <-> CC Outputs/Current setpoint value Ch.2
//     PlcTask Outputs/GVL_iXlinker.EtherCAT_Master_ATxxxx.Beckhoff_AT1xxx.Beckhoff_AT2xxxEK1122.A_0008_AT2000_0250_0020.CC_Outputs.Current_setpoint_value_Ch[2] <-> CC Outputs/Current setpoint value Ch.3
//     PlcTask Outputs/GVL_iXlinker.EtherCAT_Master_ATxxxx.Beckhoff_AT1xxx.Beckhoff_AT2xxxEK1122.A_0008_AT2000_0250_0020.CC_Outputs.Current_setpoint_value_Ch[3] <-> CC Outputs/Current setpoint value Ch.4
//     PlcTask Outputs/GVL_iXlinker.EtherCAT_Master_ATxxxx.Beckhoff_AT1xxx.Beckhoff_AT2xxxEK1122.A_0008_AT2000_0250_0020.CC_Outputs.Current_setpoint_value_Ch[4] <-> CC Outputs/Current setpoint value Ch.5
//     PlcTask Outputs/GVL_iXlinker.EtherCAT_Master_ATxxxx.Beckhoff_AT1xxx.Beckhoff_AT2xxxEK1122.A_0008_AT2000_0250_0020.CC_Outputs.Current_setpoint_value_Ch[5] <-> CC Outputs/Current setpoint value Ch.6
//     PlcTask Outputs/GVL_iXlinker.EtherCAT_Master_ATxxxx.Beckhoff_AT1xxx.Beckhoff_AT2xxxEK1122.A_0008_AT2000_0250_0020.CC_Outputs.Current_setpoint_value_Ch[6] <-> CC Outputs/Current setpoint value Ch.7
//     PlcTask Outputs/GVL_iXlinker.EtherCAT_Master_ATxxxx.Beckhoff_AT1xxx.Beckhoff_AT2xxxEK1122.A_0008_AT2000_0250_0020.CC_Outputs.Current_setpoint_value_Ch[7] <-> CC Outputs/Current setpoint value Ch.8
//     PlcTask Outputs/GVL_iXlinker.EtherCAT_Master_ATxxxx.Beckhoff_AT1xxx.Beckhoff_AT2xxxEK1122.A_0008_AT2000_0250_0020.CC_Outputs.Current_setpoint_value_Ch[8] <-> CC Outputs/Current setpoint value Ch.9
//     PlcTask Outputs/GVL_iXlinker.EtherCAT_Master_ATxxxx.Beckhoff_AT1xxx.Beckhoff_AT2xxxEK1122.A_0008_AT2000_0250_0020.CC_Outputs.Current_setpoint_value_Ch[9] <-> CC Outputs/Current setpoint value Ch.10
//     PlcTask Outputs/GVL_iXlinker.EtherCAT_Master_ATxxxx.Beckhoff_AT1xxx.Beckhoff_AT2xxxEK1122.A_0008_AT2000_0250_0020.CC_Outputs.Current_setpoint_value_Ch[10] <-> CC Outputs/Current setpoint value Ch.11
//     PlcTask Outputs/GVL_iXlinker.EtherCAT_Master_ATxxxx.Beckhoff_AT1xxx.Beckhoff_AT2xxxEK1122.A_0008_AT2000_0250_0020.CC_Outputs.Current_setpoint_value_Ch[11] <-> CC Outputs/Current setpoint value Ch.12
//     PlcTask Outputs/GVL_iXlinker.EtherCAT_Master_ATxxxx.Beckhoff_AT1xxx.Beckhoff_AT2xxxEK1122.A_0008_AT2000_0250_0020.CC_Outputs.Current_setpoint_value_Ch[12] <-> CC Outputs/Current setpoint value Ch.13
//     PlcTask Outputs/GVL_iXlinker.EtherCAT_Master_ATxxxx.Beckhoff_AT1xxx.Beckhoff_AT2xxxEK1122.A_0008_AT2000_0250_0020.CC_Outputs.Current_setpoint_value_Ch[13] <-> CC Outputs/Current setpoint value Ch.14
//     PlcTask Outputs/GVL_iXlinker.EtherCAT_Master_ATxxxx.Beckhoff_AT1xxx.Beckhoff_AT2xxxEK1122.A_0008_AT2000_0250_0020.CC_Outputs.Current_setpoint_value_Ch[14] <-> CC Outputs/Current setpoint value Ch.15
//     PlcTask Inputs/GVL_iXlinker.EtherCAT_Master_ATxxxx.Beckhoff_AT1xxx.Beckhoff_AT2xxxEK1122.A_0008_AT2000_0250_0020.WcState.WcState <-> WcState/WcState
//     PlcTask Inputs/GVL_iXlinker.EtherCAT_Master_ATxxxx.Beckhoff_AT1xxx.Beckhoff_AT2xxxEK1122.A_0008_AT2000_0250_0020.WcState.InputToggle <-> WcState/InputToggle
//     PlcTask Inputs/GVL_iXlinker.EtherCAT_Master_ATxxxx.Beckhoff_AT1xxx.Beckhoff_AT2xxxEK1122.A_0008_AT2000_0250_0020.InfoData.AdsAddr <-> InfoData/AdsAddr
//     PlcTask Inputs/GVL_iXlinker.EtherCAT_Master_ATxxxx.Beckhoff_AT1xxx.Beckhoff_AT2xxxEK1122.A_0008_AT2000_0250_0020.InfoData.DcOutputShift <-> InfoData/DcOutputShift
//     PlcTask Inputs/GVL_iXlinker.EtherCAT_Master_ATxxxx.Beckhoff_AT1xxx.Beckhoff_AT2xxxEK1122.A_0008_AT2000_0250_0020.InfoData.DcInputShift <-> InfoData/DcInputShift
//     PlcTask Inputs/GVL_iXlinker.EtherCAT_Master_ATxxxx.Beckhoff_AT1xxx.Beckhoff_AT2xxxEK1122.A_0008_AT2000_0250_0020.InfoData.State <-> InfoData/State
//   PLC/PLC Instance <-> EtherCAT Master ATxxxx/Beckhoff AT1xxx/Beckhoff AT2xxxEK1122/A_0009(AT2000-0250-0021)
//     PlcTask Inputs/GVL_iXlinker.EtherCAT_Master_ATxxxx.Beckhoff_AT1xxx.Beckhoff_AT2xxxEK1122.A_0009_AT2000_0250_0021.CC_Inputs.Status <-> CC Inputs/Status
//     PlcTask Inputs/GVL_iXlinker.EtherCAT_Master_ATxxxx.Beckhoff_AT1xxx.Beckhoff_AT2xxxEK1122.A_0009_AT2000_0250_0021.CC_Inputs.Current_actual_value_Ch[0] <-> CC Inputs/Current actual value Ch.1
//     PlcTask Inputs/GVL_iXlinker.EtherCAT_Master_ATxxxx.Beckhoff_AT1xxx.Beckhoff_AT2xxxEK1122.A_0009_AT2000_0250_0021.CC_Inputs.Current_actual_value_Ch[1] <-> CC Inputs/Current actual value Ch.2
//     PlcTask Inputs/GVL_iXlinker.EtherCAT_Master_ATxxxx.Beckhoff_AT1xxx.Beckhoff_AT2xxxEK1122.A_0009_AT2000_0250_0021.CC_Inputs.Current_actual_value_Ch[2] <-> CC Inputs/Current actual value Ch.3
//     PlcTask Inputs/GVL_iXlinker.EtherCAT_Master_ATxxxx.Beckhoff_AT1xxx.Beckhoff_AT2xxxEK1122.A_0009_AT2000_0250_0021.CC_Inputs.Current_actual_value_Ch[3] <-> CC Inputs/Current actual value Ch.4
//     PlcTask Inputs/GVL_iXlinker.EtherCAT_Master_ATxxxx.Beckhoff_AT1xxx.Beckhoff_AT2xxxEK1122.A_0009_AT2000_0250_0021.CC_Inputs.Current_actual_value_Ch[4] <-> CC Inputs/Current actual value Ch.5
//     PlcTask Inputs/GVL_iXlinker.EtherCAT_Master_ATxxxx.Beckhoff_AT1xxx.Beckhoff_AT2xxxEK1122.A_0009_AT2000_0250_0021.CC_Inputs.Current_actual_value_Ch[5] <-> CC Inputs/Current actual value Ch.6
//     PlcTask Inputs/GVL_iXlinker.EtherCAT_Master_ATxxxx.Beckhoff_AT1xxx.Beckhoff_AT2xxxEK1122.A_0009_AT2000_0250_0021.CC_Inputs.Current_actual_value_Ch[6] <-> CC Inputs/Current actual value Ch.7
//     PlcTask Inputs/GVL_iXlinker.EtherCAT_Master_ATxxxx.Beckhoff_AT1xxx.Beckhoff_AT2xxxEK1122.A_0009_AT2000_0250_0021.CC_Inputs.Current_actual_value_Ch[7] <-> CC Inputs/Current actual value Ch.8
//     PlcTask Inputs/GVL_iXlinker.EtherCAT_Master_ATxxxx.Beckhoff_AT1xxx.Beckhoff_AT2xxxEK1122.A_0009_AT2000_0250_0021.CC_Inputs.Current_actual_value_Ch[8] <-> CC Inputs/Current actual value Ch.9
//     PlcTask Inputs/GVL_iXlinker.EtherCAT_Master_ATxxxx.Beckhoff_AT1xxx.Beckhoff_AT2xxxEK1122.A_0009_AT2000_0250_0021.CC_Inputs.Current_actual_value_Ch[9] <-> CC Inputs/Current actual value Ch.10
//     PlcTask Inputs/GVL_iXlinker.EtherCAT_Master_ATxxxx.Beckhoff_AT1xxx.Beckhoff_AT2xxxEK1122.A_0009_AT2000_0250_0021.CC_Inputs.Current_actual_value_Ch[10] <-> CC Inputs/Current actual value Ch.11
//     PlcTask Inputs/GVL_iXlinker.EtherCAT_Master_ATxxxx.Beckhoff_AT1xxx.Beckhoff_AT2xxxEK1122.A_0009_AT2000_0250_0021.CC_Inputs.Current_actual_value_Ch[11] <-> CC Inputs/Current actual value Ch.12
//     PlcTask Inputs/GVL_iXlinker.EtherCAT_Master_ATxxxx.Beckhoff_AT1xxx.Beckhoff_AT2xxxEK1122.A_0009_AT2000_0250_0021.CC_Inputs.Current_actual_value_Ch[12] <-> CC Inputs/Current actual value Ch.13
//     PlcTask Inputs/GVL_iXlinker.EtherCAT_Master_ATxxxx.Beckhoff_AT1xxx.Beckhoff_AT2xxxEK1122.A_0009_AT2000_0250_0021.CC_Inputs.Current_actual_value_Ch[13] <-> CC Inputs/Current actual value Ch.14
//     PlcTask Inputs/GVL_iXlinker.EtherCAT_Master_ATxxxx.Beckhoff_AT1xxx.Beckhoff_AT2xxxEK1122.A_0009_AT2000_0250_0021.CC_Inputs.Current_actual_value_Ch[14] <-> CC Inputs/Current actual value Ch.15
//     PlcTask Outputs/GVL_iXlinker.EtherCAT_Master_ATxxxx.Beckhoff_AT1xxx.Beckhoff_AT2xxxEK1122.A_0009_AT2000_0250_0021.CC_Outputs.Control <-> CC Outputs/Control
//     PlcTask Outputs/GVL_iXlinker.EtherCAT_Master_ATxxxx.Beckhoff_AT1xxx.Beckhoff_AT2xxxEK1122.A_0009_AT2000_0250_0021.CC_Outputs.Current_setpoint_value_Ch[0] <-> CC Outputs/Current setpoint value Ch.1
//     PlcTask Outputs/GVL_iXlinker.EtherCAT_Master_ATxxxx.Beckhoff_AT1xxx.Beckhoff_AT2xxxEK1122.A_0009_AT2000_0250_0021.CC_Outputs.Current_setpoint_value_Ch[1] <-> CC Outputs/Current setpoint value Ch.2
//     PlcTask Outputs/GVL_iXlinker.EtherCAT_Master_ATxxxx.Beckhoff_AT1xxx.Beckhoff_AT2xxxEK1122.A_0009_AT2000_0250_0021.CC_Outputs.Current_setpoint_value_Ch[2] <-> CC Outputs/Current setpoint value Ch.3
//     PlcTask Outputs/GVL_iXlinker.EtherCAT_Master_ATxxxx.Beckhoff_AT1xxx.Beckhoff_AT2xxxEK1122.A_0009_AT2000_0250_0021.CC_Outputs.Current_setpoint_value_Ch[3] <-> CC Outputs/Current setpoint value Ch.4
//     PlcTask Outputs/GVL_iXlinker.EtherCAT_Master_ATxxxx.Beckhoff_AT1xxx.Beckhoff_AT2xxxEK1122.A_0009_AT2000_0250_0021.CC_Outputs.Current_setpoint_value_Ch[4] <-> CC Outputs/Current setpoint value Ch.5
//     PlcTask Outputs/GVL_iXlinker.EtherCAT_Master_ATxxxx.Beckhoff_AT1xxx.Beckhoff_AT2xxxEK1122.A_0009_AT2000_0250_0021.CC_Outputs.Current_setpoint_value_Ch[5] <-> CC Outputs/Current setpoint value Ch.6
//     PlcTask Outputs/GVL_iXlinker.EtherCAT_Master_ATxxxx.Beckhoff_AT1xxx.Beckhoff_AT2xxxEK1122.A_0009_AT2000_0250_0021.CC_Outputs.Current_setpoint_value_Ch[6] <-> CC Outputs/Current setpoint value Ch.7
//     PlcTask Outputs/GVL_iXlinker.EtherCAT_Master_ATxxxx.Beckhoff_AT1xxx.Beckhoff_AT2xxxEK1122.A_0009_AT2000_0250_0021.CC_Outputs.Current_setpoint_value_Ch[7] <-> CC Outputs/Current setpoint value Ch.8
//     PlcTask Outputs/GVL_iXlinker.EtherCAT_Master_ATxxxx.Beckhoff_AT1xxx.Beckhoff_AT2xxxEK1122.A_0009_AT2000_0250_0021.CC_Outputs.Current_setpoint_value_Ch[8] <-> CC Outputs/Current setpoint value Ch.9
//     PlcTask Outputs/GVL_iXlinker.EtherCAT_Master_ATxxxx.Beckhoff_AT1xxx.Beckhoff_AT2xxxEK1122.A_0009_AT2000_0250_0021.CC_Outputs.Current_setpoint_value_Ch[9] <-> CC Outputs/Current setpoint value Ch.10
//     PlcTask Outputs/GVL_iXlinker.EtherCAT_Master_ATxxxx.Beckhoff_AT1xxx.Beckhoff_AT2xxxEK1122.A_0009_AT2000_0250_0021.CC_Outputs.Current_setpoint_value_Ch[10] <-> CC Outputs/Current setpoint value Ch.11
//     PlcTask Outputs/GVL_iXlinker.EtherCAT_Master_ATxxxx.Beckhoff_AT1xxx.Beckhoff_AT2xxxEK1122.A_0009_AT2000_0250_0021.CC_Outputs.Current_setpoint_value_Ch[11] <-> CC Outputs/Current setpoint value Ch.12
//     PlcTask Outputs/GVL_iXlinker.EtherCAT_Master_ATxxxx.Beckhoff_AT1xxx.Beckhoff_AT2xxxEK1122.A_0009_AT2000_0250_0021.CC_Outputs.Current_setpoint_value_Ch[12] <-> CC Outputs/Current setpoint value Ch.13
//     PlcTask Outputs/GVL_iXlinker.EtherCAT_Master_ATxxxx.Beckhoff_AT1xxx.Beckhoff_AT2xxxEK1122.A_0009_AT2000_0250_0021.CC_Outputs.Current_setpoint_value_Ch[13] <-> CC Outputs/Current setpoint value Ch.14
//     PlcTask Outputs/GVL_iXlinker.EtherCAT_Master_ATxxxx.Beckhoff_AT1xxx.Beckhoff_AT2xxxEK1122.A_0009_AT2000_0250_0021.CC_Outputs.Current_setpoint_value_Ch[14] <-> CC Outputs/Current setpoint value Ch.15
//     PlcTask Inputs/GVL_iXlinker.EtherCAT_Master_ATxxxx.Beckhoff_AT1xxx.Beckhoff_AT2xxxEK1122.A_0009_AT2000_0250_0021.WcState.WcState <-> WcState/WcState
//     PlcTask Inputs/GVL_iXlinker.EtherCAT_Master_ATxxxx.Beckhoff_AT1xxx.Beckhoff_AT2xxxEK1122.A_0009_AT2000_0250_0021.WcState.InputToggle <-> WcState/InputToggle
//     PlcTask Inputs/GVL_iXlinker.EtherCAT_Master_ATxxxx.Beckhoff_AT1xxx.Beckhoff_AT2xxxEK1122.A_0009_AT2000_0250_0021.InfoData.AdsAddr <-> InfoData/AdsAddr
//     PlcTask Inputs/GVL_iXlinker.EtherCAT_Master_ATxxxx.Beckhoff_AT1xxx.Beckhoff_AT2xxxEK1122.A_0009_AT2000_0250_0021.InfoData.DcOutputShift <-> InfoData/DcOutputShift
//     PlcTask Inputs/GVL_iXlinker.EtherCAT_Master_ATxxxx.Beckhoff_AT1xxx.Beckhoff_AT2xxxEK1122.A_0009_AT2000_0250_0021.InfoData.DcInputShift <-> InfoData/DcInputShift
//     PlcTask Inputs/GVL_iXlinker.EtherCAT_Master_ATxxxx.Beckhoff_AT1xxx.Beckhoff_AT2xxxEK1122.A_0009_AT2000_0250_0021.InfoData.State <-> InfoData/State
